REGION Network 3: Block description — Sections 4 to 10
   // ▄▄▄▄▄▄▄▄▄▄▄▄▄▄▄▄▄▄▄▄▄▄▄▄▄▄▄▄▄▄▄▄▄▄▄▄▄▄▄▄▄▄▄▄
   // 4.     Supervisory system interface
   // 
   // 
   // There is no supervisory system interface for this block. It is a debug simulation module and as 
   // such has no graphical symbol, block icon or faceplate.
   // 
   // 
   //                ━━━   ⬙⬙⬙⬙⬙⬙   ━━━
   // 
   // 
   // 
   // ▄▄▄▄▄▄▄▄▄▄▄▄▄▄▄▄▄▄▄▄▄▄▄▄▄▄▄▄▄▄▄▄▄▄▄▄▄▄▄▄▄▄▄▄
   // 5.     PARAMETERS
   // 
   // 
   // The following parameters are associated with the block:
   // 
   //  
   //  ――――――――――――――――――――――――――――――――――――――――――
   //  PARAM         FUNCTION                    TYPE      IN-OUT 
   //  ――――――――――――――――――――――――――――――――――――――――――
   //  SYS_SIGNALS      Common system signals              UT21000    In
   //           logic and timing signals for parametric access
   // 
   //  TRIGGER       Activates the simulation (the simulation will run     Bool      In
   //           whilever this signal is high), the elapsed time 
   //           is measured from the rising edge of this signal
   // 
   //  INPUT        The input time function, x(t) in the calculations     Real      In
   // 
   //  DYNAMIC_DATA      Data structure that holds the live data for the       UT39511    InOut
   //           simulation (damping factor, natural frequency, 
   //           system gain, elapsed time &c.)
   // 
   //  OUTPUT       The output time response, y(t) in the calculations   Real      Out
   //  ――――――――――――――――――――――――――――――――――――――――――
   // 
   //                ━━━   ⬙⬙⬙⬙⬙⬙   ━━━
   // 
   // 
   // 
   // ▄▄▄▄▄▄▄▄▄▄▄▄▄▄▄▄▄▄▄▄▄▄▄▄▄▄▄▄▄▄▄▄▄▄▄▄▄▄▄▄▄▄▄▄
   // 6.     DATA STRUCTURES AND USAGE
   // 
   // 
   // The block has the following associated data structure:
   // 
   // 
   //  ――――――――――――――――――――――――――――――――――――――――――
   //  DATA STRUCTURE             DESCRIPTION
   //  ――――――――――――――――――――――――――――――――――――――――――
   //  UT01000_St_SysRevision          Revision information for this block    See FC01001
   //  UT01001_St_SysLicence           Licence information for this block  See FC01001
   //  UT21000_Dy_SysSignals           System signals for logic and timing  See FC01001
   // 
   //  UT39511_Dy_DebugInst1Order        Dynamic data storage, contains live data, such as 
   //                     calculation variables, elapsed time, oscillation 
   //                     frequency and status signals
   //  ――――――――――――――――――――――――――――――――――――――――――
   // 
   // 
   // ▂▂▂▂▂▂▂▂▂▂▂▂▂▂▂▂▂▂▂▂▂▂▂▂▂▂▂▂▂▂▂▂▂▂▂▂▂▂▂▂▂▂▂▂
   // 6.1      UT39511_Dy_DebugInst1Order
   // 
   // The static data structure for an isolating valve.
   // 
   // 
   // 
   //  UT39511_Dy_DebugInst1Order (full contents)
   //  ――――――――――――――――――――――――――――――――――――――――――
   //  SIGNAL NAME          FUNCTION                     TYPE
   //  ――――――――――――――――――――――――――――――――――――――――――
   //  k_Gain             CONSTANT — Simulation system gain        Real
   //  k_TimeConstant        CONSTANT — The system time constant τ (s)       Real
   // 
   //  status_Running      STATUS — Simulation is running  Bool
   //                      (1 = running, 0 = stopped)
   //  status_Stopped        STATUS — Simulation is stopped (not running)    Bool
   //                      (1 = stopped, 0 = running)
   //  status_SteadyState     STATUS — Response is at steady state value             Bool
   //                      (1 = stead state reached ±2%)
   //  status_Aut           STATUS — Simulation is in automatic mode      Bool
   //                      (1 = automatic, 0 = manual)
   //  status_Man          STATUS — Simulation is in manual mode        Bool
   //                      (1 = manual, 0 = automatic)
   // 
   //  cal_TimeSteady        CALC — Time to reach steady state (s)       Real
   //                    zero for unstable response
   // 
   //  mode_AutMan       MODE — Automatic/manual mode selection     Bool
   //                      (1 = auto mode, 0 = manual mode)
   //  mode_ManTime       MODE — Manual mode time value (s)        Real
   // 
   //  actual_Output       ACTUAL — Output signal, same as OUTPUT param    Real
   //                      (y(t) or y[n])
   //  actual_PrevOutput      ACTUAL — Output value from the previous iteration    Real
   //                      (y[n-1])
   //  actual_StartTime         ACTUAL — CPU time when simulation started       DTL
   //  actual_Time        ACTUAL — CPU time of this iteration of simulation  DTL
   //  actual_PrevTime       ACTUAL — CPU time of last iteration of simulation     DTL
   //  actual_RunTime        ACTUAL — Elapsed time since the            Real
   //                      simulation started (s)
   //  actual_DeltaTime        ACTUAL — Time between this and last iteration (s)   Real
   //  ――――――――――――――――――――――――――――――――――――――――――
   // 
   // 
   //                ━━━   ⬙⬙⬙⬙⬙⬙   ━━━
   // 
   // 
   // 
   // ▄▄▄▄▄▄▄▄▄▄▄▄▄▄▄▄▄▄▄▄▄▄▄▄▄▄▄▄▄▄▄▄▄▄▄▄▄▄▄▄▄▄▄▄
   // 7.     CONSTANTS AND TEMPORARY (LOCAL) DATA
   // 
   // 
   // 
   // ▂▂▂▂▂▂▂▂▂▂▂▂▂▂▂▂▂▂▂▂▂▂▂▂▂▂▂▂▂▂▂▂▂▂▂▂▂▂▂▂▂▂▂▂
   // 7.1     Constants
   // 
   // 
   // The following constants data is used:
   // 
   //  ――――――――――――――――――――――――――――――――――――――――――
   //  SIGNAL NAME       Value     FUNCTION                 TYPE
   //  ――――――――――――――――――――――――――――――――――――――――――
   //  k_NEG_MAX       3.4E-38    Largest negative REAL number         Real
   //  ――――――――――――――――――――――――――――――――――――――――――
   // 
   // 
   // 
   // ▂▂▂▂▂▂▂▂▂▂▂▂▂▂▂▂▂▂▂▂▂▂▂▂▂▂▂▂▂▂▂▂▂▂▂▂▂▂▂▂▂▂▂▂
   // 7.2     Temporary (local) data
   // 
   // 
   // The following temporary data is used:
   // 
   //  ――――――――――――――――――――――――――――――――――――――――――
   //  SIGNAL NAME          FUNCTION                  TYPE
   //  ――――――――――――――――――――――――――――――――――――――――――
   //  revInfo             Revision information for the block         UT01000
   //  licInfo           Licensing information for the block      UT01001
   //  act_CPUTime           Current CPU time (this block call)       DTL
   //  cal_01          Partial calculation see § 3.4 for details      Real
   //  cal_02          Partial calculation see § 3.4 for details      Real
   //  cal_03          Partial calculation see § 3.4 for details      Real
   //  cal_04          Partial calculation see § 3.4 for details      Real
   //  cal_05          Partial calculation see § 3.4 for details      Real
   //  cal_06          Partial calculation see § 3.4 for details      Real
   //  wrkElapsedTime          Working storage area (current elapsed time)    LTIme
   //  wrkDeltaTime         Working storage area (current delta time)   LTIme
   //  wrkInt           Working storage area (integer)          Int
   //  wrkLInt            Working storage area (long integer)        ULInt
   //  wrkReal           Working storage (Real)             Real
   //  ――――――――――――――――――――――――――――――――――――――――――
   // 
   // 
   //                ━━━   ⬙⬙⬙⬙⬙⬙   ━━━
   // 
   // 
   // 
   // ▄▄▄▄▄▄▄▄▄▄▄▄▄▄▄▄▄▄▄▄▄▄▄▄▄▄▄▄▄▄▄▄▄▄▄▄▄▄▄▄▄▄▄▄
   // 8.     BLOCK CALLS AND ASSOCIATIONS
   // 
   // 
   // This section details any blocks which may be called from within this software module (subroutine 
   // functions for example), any partner blocks with which it may be associated (for example a 
   // receive module that is partner with a transmit module &c.). It lists any system functions which 
   // may be called (e.g. reading the real time clock) and any system data types that may be used.
   // 
   // Finally, it lists any special calling requirements for the block (for example, must be called from 
   // within a cyclic interrupt organisation block) and if the block is using “optimised access” (this is 
   // the default arrangement).
   // 
   // 
   // 
   // ▂▂▂▂▂▂▂▂▂▂▂▂▂▂▂▂▂▂▂▂▂▂▂▂▂▂▂▂▂▂▂▂▂▂▂▂▂▂▂▂▂▂▂▂
   // 8.1     Block calls from within this module
   // 
   // 
   // There are no PAL block calls from within this block.
   // 
   // 
   // 
   // ▂▂▂▂▂▂▂▂▂▂▂▂▂▂▂▂▂▂▂▂▂▂▂▂▂▂▂▂▂▂▂▂▂▂▂▂▂▂▂▂▂▂▂▂
   // 8.2     Blocks associated with this module
   // 
   // 
   // This is a stand-alone block and is not associated with any other blocks.
   // 
   // 
   // 
   // ▂▂▂▂▂▂▂▂▂▂▂▂▂▂▂▂▂▂▂▂▂▂▂▂▂▂▂▂▂▂▂▂▂▂▂▂▂▂▂▂▂▂▂▂
   // 8.3     System block calls and system data types
   // 
   // The following calls are made to system blocks:
   // 
   // 
   //  System block calls
   //  ――――――――――――――――――――――――――――――――――――――――――
   //  BLOCK          TITLE             DESCRIPTION  
   //  ――――――――――――――――――――――――――――――――――――――――――
   //  RD_LOC_T             Read the local RTC time    Reads the CPU real time clock 
   //  ――――――――――――――――――――――――――――――――――――――――――
   // 
   // There are no special system data types used.
   // 
   // 
   //                ━━━   ⬙⬙⬙⬙⬙⬙   ━━━
   // 
   // 
   // 
   // ▂▂▂▂▂▂▂▂▂▂▂▂▂▂▂▂▂▂▂▂▂▂▂▂▂▂▂▂▂▂▂▂▂▂▂▂▂▂▂▂▂▂▂▂
   // 8.4     Special properties and requirements
   // 
   // 
   // 
   // ▁▁▁▁▁▁▁▁▁▁▁▁▁▁▁▁▁▁▁▁▁▁▁▁▁▁▁▁▁▁▁▁▁▁▁▁▁▁▁▁▁▁▁▁
   // 8.4.1     Block optimisation, IEC compatibility and library conformance
   // 
   // 
   //    •   Block optimisation is ACTIVE for this block.
   // 
   //    •   The block has been checked for IEC compatibility and is compliant.
   // 
   //    •   The block is compatible with all IEC library-conformance module constraints
   // 
   // 
   // 
   // ▁▁▁▁▁▁▁▁▁▁▁▁▁▁▁▁▁▁▁▁▁▁▁▁▁▁▁▁▁▁▁▁▁▁▁▁▁▁▁▁▁▁▁▁
   // 8.4.2     Calling requirements
   // 
   // 
   // There are no special calling requirements for this block.
   // 
   //                ━━━   ⬙⬙⬙⬙⬙⬙   ━━━
   // 
   // 
   // 
   // ▄▄▄▄▄▄▄▄▄▄▄▄▄▄▄▄▄▄▄▄▄▄▄▄▄▄▄▄▄▄▄▄▄▄▄▄▄▄▄▄▄▄▄▄
   // 9.     EXAMPLE USAGE
   // 
   // 
   // The following shows a typical deployment of FC19512:
   // 
   //                         ┌─────────────
   //      ───────────────────┤ FC19511
   //                         ├───────────────┤
   //    "DB21001_DY_StdGlobalData".SysSignals ─┤ SYS_SIGNALS                  %MD910 
   //                         │               OUTPUT ├─  "SIM001_OUTPUT"
   //                         │               │
   //                                                        "1.0" ─┤ INPUT                     │
   //                         │               │
   //                   %M999.0     │               │
   //                  "SIM001_TRIG" ─┤ TRIGGER                     │
   //                         │               │
   //                         │
   //      "DB39511_Dy_DebugInst1Order".SIM001 ─┤ DYNAMIC_DATA
   //                         │
   //                         │
   //                                         │
   //                                ─────────┘
   // 
   // 
   //               ━━━   ⬙⬙⬙⬙⬙⬙   ━━━
   // 
   // 
   // 
   // ▄▄▄▄▄▄▄▄▄▄▄▄▄▄▄▄▄▄▄▄▄▄▄▄▄▄▄▄▄▄▄▄▄▄▄▄▄▄▄▄▄▄▄▄
   // 10.     TEST AND VERIFICATION PATH
   // 
   // 
   // The following diagram shows the full test and verification path for the formal release of each 
   // version of the software module. See the Test Plan [Ref. 003] for full details, available here:
   //         https://psop.uk/pal-tp-p
   // 
   // 
   //         FC19151-T001
   // 
   //     Test version: 000.801  
   //  Released version: 001.000   
   // Released commit: D0017    
   // 
   //        SCR      SMT 
   // ＿＿＿＿＿＿┌┐＿＿ ▛▜ ＿
   //       └┘   ▙▟  
   // Initial test           
   // 
   // Initial test to release the      
   // module following the      
   // development stage.       
   // Full SMT              
   // 
   // 
   // Where:
   // ――――――――――――――――――――――――――――――――――――――――――――
   //  SCR    Source Code Review      A visual inspection of the software to ensure it has been written  
   // ┌┐             to the correct standards, uses the correct structures within the
   // └┘             software and is generally suitable for deployment.               
   // 
   //  SMT Software Module Test    A full and detailed test of an individual software module in
   //   ▛▜              isolation; such testing requires that all branches of the 
   //   ▙▟              software are tested. 
   // 
   //                It tests all the interfaces to the module, any data recorded or 
   //                stored by the module, all error and exception handling functions 
   //                and tests all timed and interrupt driven operations.
   // 
   //  SCV Software Compatibility     A mechanism for verifying that no executable code software 
   // ╓╖    Verification          changes have been made to a module following changes to
   // ╙╜             comment fields.
   // 
   //                Allows typographical errors &c. to be corrected without forcing 
   //                a full SMT on a module that has not functionally changed.
   // ――――――――――――――――――――――――――――――――――――――――――――
   // 
   // An SCV can only be performed on a module that has at some point previously, successfully 
   // completed both an SCR and SMT. Where an SCV is implemented, it replaces the requirement for 
   // both the SCR and the SMT for the test iteration in question.
   // 
   //                ━━━   ⬙⬙⬙⬙⬙⬙   ━━━
   // 
   // 
   // ██████████████ █ █ █ █  END   █ █ █ █ ██████████████
END_REGION

REGION Network 4: Current revision and modification history
   // ▄▄▄▄▄▄▄▄▄▄▄▄▄▄▄▄▄▄▄▄▄▄▄▄▄▄▄▄▄▄▄▄▄▄▄▄▄▄▄▄▄▄▄▄
   // MODIFICATION HISTORY
   // 
   // 
   // The revision data shown here, in the network comments, contains additional information 
   // reflecting the software development workflow under the version control system (VCS) employed 
   // to track all software changes.
   // 
   // The VCS in use is the Git Source Code Management system in conjunction with the GitHub online 
   // hosting system. The software in its entirety is available in the GitHub remote repository:
   // 
   //      https://github.com/practicalseries/PS2001-pal-software
   // 
   // The repository is public and can be freely copied (forked in GitHub terminology) and used 
   // under the MIT licence. 
   // 
   // The MIT licence is reproduced in full in the last network of this software module.
   // 
   // 
   //  ―――――――――――――――――――――――――――――――――――――――――――
   //  DATE       REVISION             MASTER BRANCH     DEV
   //          (nnn.amm)   COMMIT TAG    (Base ---> Merge)    BRANCH   Author
   //  ———————————————————————————————————————————
   //  2023.02.26    000.101   D0016A-000.101   D0016 N/A     D0016A   M. Gledhill
   //                        FC19511 Block created — Comments added
   //  ———————————————————————————————————————————
   //   Where: nnn  =  Major revision
   //         a  =  Type (1-7 Development, 8 Proving, 9 Qualification, 0 Release)
   //       mm  =  Minor revision (must be 00 if a = 0)
   //         Block properties version number should be set to nn.a (only one decimal place)
   // 
   // ▄▄▄▄▄▄▄▄▄▄▄▄▄▄▄▄▄▄▄▄▄▄▄▄▄▄▄▄▄▄▄▄▄▄▄▄▄▄▄▄▄▄▄▄
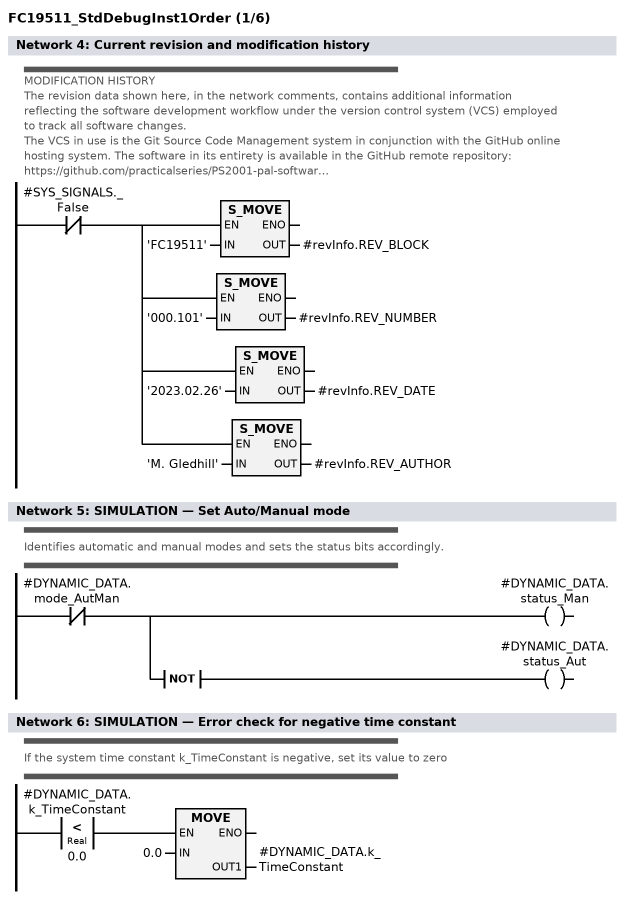
   RUNG wire#powerrail
      I_Contact( #SYS_SIGNALS._False )
      wire#w1
      S_Move(in := 'FC19511', out => #revInfo.REV_BLOCK)
   END_RUNG
   RUNG wire#w1
      S_Move(in := '000.101', out => #revInfo.REV_NUMBER)
   END_RUNG
   RUNG wire#w1
      S_Move(in := '2023.02.26', out => #revInfo.REV_DATE)
   END_RUNG
   RUNG wire#w1
      S_Move(in := 'M. Gledhill', out => #revInfo.REV_AUTHOR)
   END_RUNG
   // the same network as SCL:
   IF NOT #SYS_SIGNALS._False THEN
       #revInfo.REV_BLOCK := 'FC19511';
       #revInfo.REV_NUMBER := '000.101';
       #revInfo.REV_DATE := '2023.02.26';
       #revInfo.REV_AUTHOR := 'M. Gledhill';
   END_IF;
END_REGION

REGION Network 5: SIMULATION — Set Auto/Manual mode
   // ▀▀▀▀▀▀▀▀▀▀▀▀▀▀▀▀▀▀▀▀▀▀▀▀▀▀▀▀▀▀▀▀▀▀▀▀▀▀▀▀▀▀▀▀
   // Identifies automatic and manual modes and sets the status bits accordingly.
   // ▄▄▄▄▄▄▄▄▄▄▄▄▄▄▄▄▄▄▄▄▄▄▄▄▄▄▄▄▄▄▄▄▄▄▄▄▄▄▄▄▄▄▄▄
   RUNG wire#powerrail
      I_Contact( #DYNAMIC_DATA.mode_AutMan )
      wire#w1
      Coil( #DYNAMIC_DATA.status_Man )
   END_RUNG
   RUNG wire#w1
      Not()
      Coil( #DYNAMIC_DATA.status_Aut )
   END_RUNG
   // the same network as SCL:
   #DYNAMIC_DATA.status_Man := NOT #DYNAMIC_DATA.mode_AutMan;
   #DYNAMIC_DATA.status_Aut := NOT (NOT #DYNAMIC_DATA.mode_AutMan);
END_REGION

REGION Network 6: SIMULATION — Error check for negative time constant
   // ▀▀▀▀▀▀▀▀▀▀▀▀▀▀▀▀▀▀▀▀▀▀▀▀▀▀▀▀▀▀▀▀▀▀▀▀▀▀▀▀▀▀▀▀
   // If the system time constant k_TimeConstant is negative, set its value to zero
   // ▄▄▄▄▄▄▄▄▄▄▄▄▄▄▄▄▄▄▄▄▄▄▄▄▄▄▄▄▄▄▄▄▄▄▄▄▄▄▄▄▄▄▄▄
   RUNG wire#powerrail
      { S7_Templates := "SrcType := Real" } LT_Contact(in1 := #DYNAMIC_DATA.k_TimeConstant, in2 := 0.0)
      Move(in := 0.0, out1 => #DYNAMIC_DATA.k_TimeConstant)
   END_RUNG
   // the same network as SCL:
   IF #DYNAMIC_DATA.k_TimeConstant < 0.0 THEN #DYNAMIC_DATA.k_TimeConstant := 0.0; END_IF;
END_REGION

REGION Network 7: SIMULATION INACTIVE — Reset data — Block end
   // ▀▀▀▀▀▀▀▀▀▀▀▀▀▀▀▀▀▀▀▀▀▀▀▀▀▀▀▀▀▀▀▀▀▀▀▀▀▀▀▀▀▀▀▀
   // If the simulation is not running (TRIGGER = 0), set status to stopped and reset all calculated data
   // and status signals.
   // 
   // Set the previous time to the current CPU time (in readiness for the start of the simulation)
   // 
   // Set the OUTPUT, actual_Output and actual_PrevOutput to zero
   // 
   // If the simulation is not running, the block will terminate at this point.
   // ▄▄▄▄▄▄▄▄▄▄▄▄▄▄▄▄▄▄▄▄▄▄▄▄▄▄▄▄▄▄▄▄▄▄▄▄▄▄▄▄▄▄▄▄
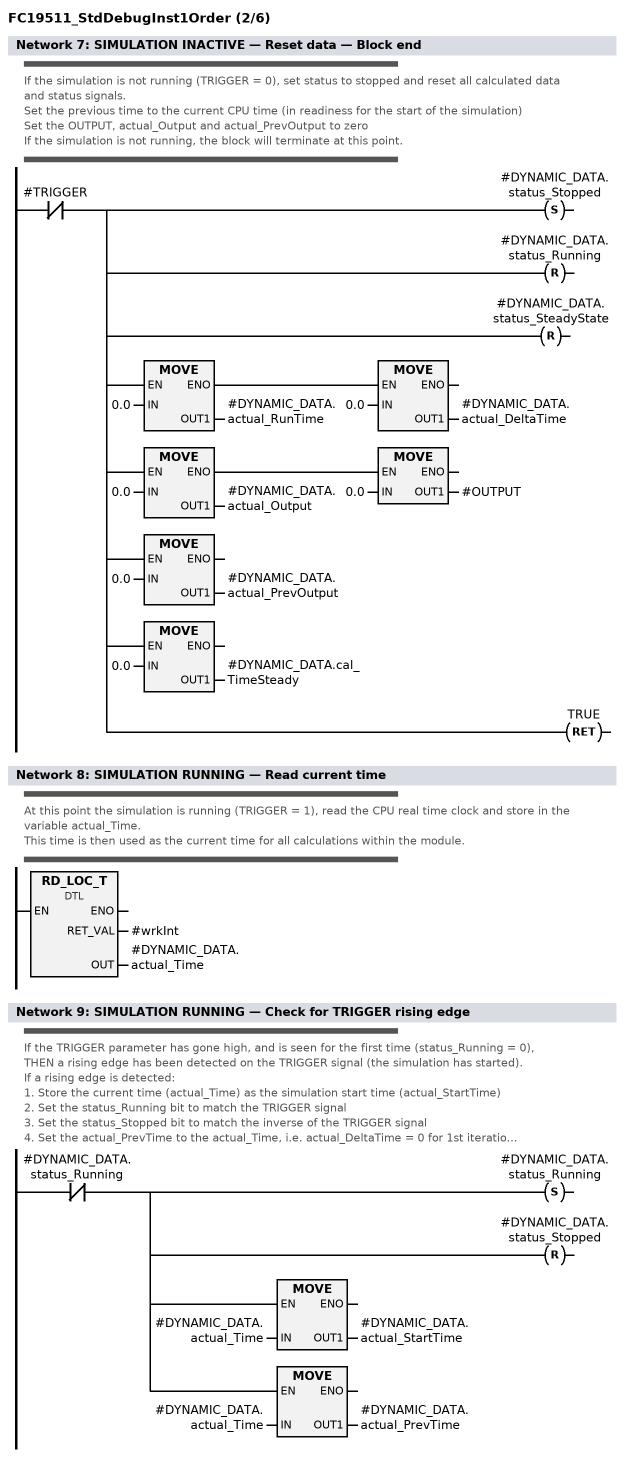
   IF NOT #TRIGGER THEN
       #DYNAMIC_DATA.status_Stopped := TRUE;
       #DYNAMIC_DATA.status_Running := FALSE;
       #DYNAMIC_DATA.status_SteadyState := FALSE;
       #DYNAMIC_DATA.actual_RunTime := 0.0;
       #DYNAMIC_DATA.actual_DeltaTime := 0.0;
       #DYNAMIC_DATA.actual_Output := 0.0;
       #OUTPUT := 0.0;
       #DYNAMIC_DATA.actual_PrevOutput := 0.0;
       #DYNAMIC_DATA.cal_TimeSteady := 0.0;
       ENO := TRUE;
       RETURN;
   END_IF;
END_REGION

REGION Network 8: SIMULATION RUNNING — Read current time
   // ▀▀▀▀▀▀▀▀▀▀▀▀▀▀▀▀▀▀▀▀▀▀▀▀▀▀▀▀▀▀▀▀▀▀▀▀▀▀▀▀▀▀▀▀
   // At this point the simulation is running (TRIGGER = 1), read the CPU real time clock and store in the 
   // variable actual_Time.
   // 
   // This time is then used as the current time for all calculations within the module.
   // ▄▄▄▄▄▄▄▄▄▄▄▄▄▄▄▄▄▄▄▄▄▄▄▄▄▄▄▄▄▄▄▄▄▄▄▄▄▄▄▄▄▄▄▄
   RUNG wire#powerrail
      { S7_Templates := "date_type := DTL" } RD_LOC_T(RET_VAL => #wrkInt, OUT => #DYNAMIC_DATA.actual_Time)
   END_RUNG
   // the same network as SCL:
   #wrkInt := RD_LOC_T(OUT => #DYNAMIC_DATA.actual_Time);
END_REGION

REGION Network 9: SIMULATION RUNNING — Check for TRIGGER rising edge
   // ▀▀▀▀▀▀▀▀▀▀▀▀▀▀▀▀▀▀▀▀▀▀▀▀▀▀▀▀▀▀▀▀▀▀▀▀▀▀▀▀▀▀▀▀
   // If the TRIGGER parameter has gone high, and is seen for the first time (status_Running = 0),
   // THEN a rising edge has been detected on the TRIGGER signal (the simulation has started).
   // 
   // If a rising edge is detected:
   //   1. Store the current time (actual_Time) as the simulation start time (actual_StartTime)
   //   2. Set the status_Running bit to match the TRIGGER signal
   //   3. Set the status_Stopped bit to match the inverse of the TRIGGER signal
   //   4. Set the actual_PrevTime to the actual_Time, i.e. actual_DeltaTime = 0 for 1st iteration
   // ▄▄▄▄▄▄▄▄▄▄▄▄▄▄▄▄▄▄▄▄▄▄▄▄▄▄▄▄▄▄▄▄▄▄▄▄▄▄▄▄▄▄▄▄
   RUNG wire#powerrail
      I_Contact( #DYNAMIC_DATA.status_Running )
      wire#w1
      S_Coil( #DYNAMIC_DATA.status_Running )
   END_RUNG
   RUNG wire#w1
      R_Coil( #DYNAMIC_DATA.status_Stopped )
   END_RUNG
   RUNG wire#w1
      Move(in := #DYNAMIC_DATA.actual_Time, out1 => #DYNAMIC_DATA.actual_StartTime)
   END_RUNG
   RUNG wire#w1
      Move(in := #DYNAMIC_DATA.actual_Time, out1 => #DYNAMIC_DATA.actual_PrevTime)
   END_RUNG
   // the same network as SCL:
   #_w1 := NOT #DYNAMIC_DATA.status_Running;
   IF #_w1 THEN
       #DYNAMIC_DATA.status_Running := TRUE;
       #DYNAMIC_DATA.status_Stopped := FALSE;
       #DYNAMIC_DATA.actual_StartTime := #DYNAMIC_DATA.actual_Time;
       #DYNAMIC_DATA.actual_PrevTime := #DYNAMIC_DATA.actual_Time;
   END_IF;
END_REGION

REGION Network 10: SIMULATION RUNNING — Calculate current elapsed time
   // ▀▀▀▀▀▀▀▀▀▀▀▀▀▀▀▀▀▀▀▀▀▀▀▀▀▀▀▀▀▀▀▀▀▀▀▀▀▀▀▀▀▀▀▀
   // If the TRIGGER parameter is high (the simulation is running), then:
   // Subtract the start time from the current time to give the current elapsed time (wrkElapsedTime)
   // 
   // The elapsed time is calculated in the LTIme format
   // ▄▄▄▄▄▄▄▄▄▄▄▄▄▄▄▄▄▄▄▄▄▄▄▄▄▄▄▄▄▄▄▄▄▄▄▄▄▄▄▄▄▄▄▄
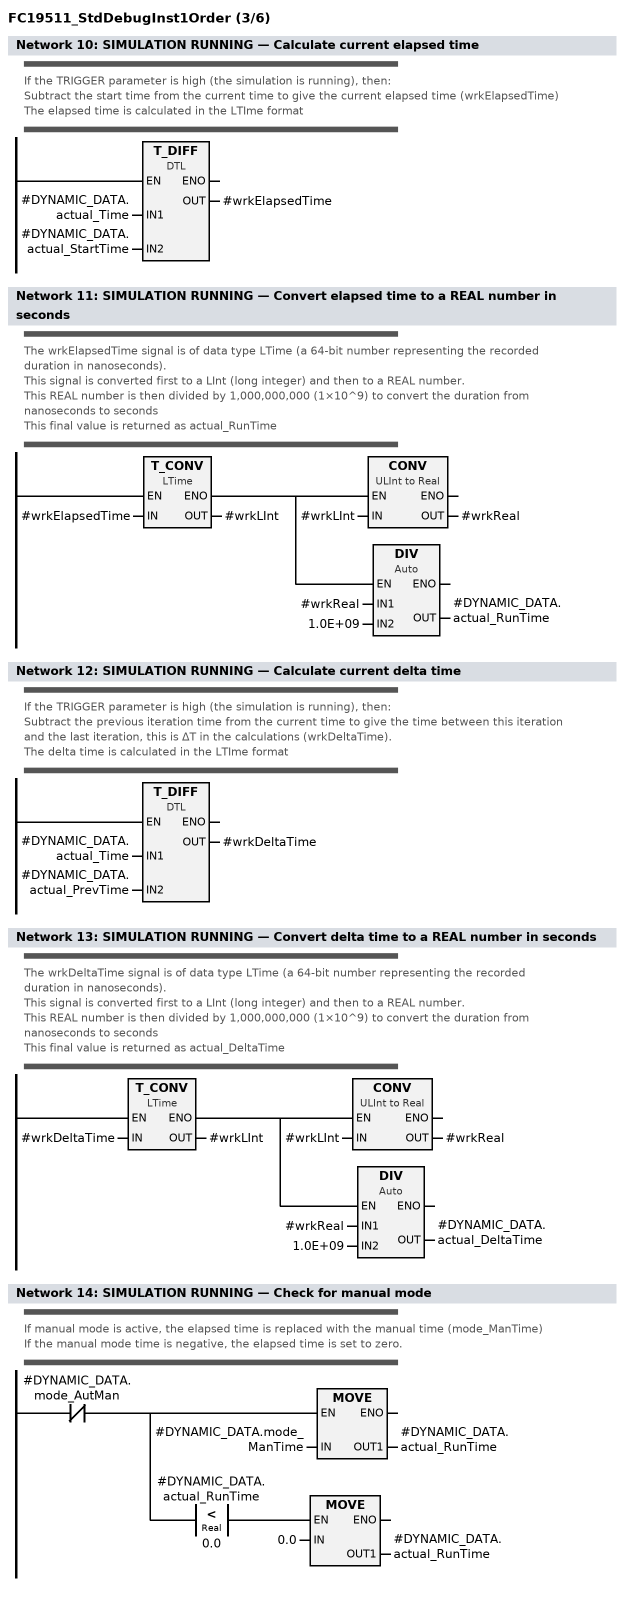
   RUNG wire#powerrail
      { S7_Templates := "[date_type := DTL, time_type := LTime]" } T_DIFF(IN1 := #DYNAMIC_DATA.actual_Time, IN2 := #DYNAMIC_DATA.actual_StartTime, OUT => #wrkElapsedTime)
   END_RUNG
   // the same network as SCL:
   T_DIFF(IN1 := #DYNAMIC_DATA.actual_Time, IN2 := #DYNAMIC_DATA.actual_StartTime, OUT => #wrkElapsedTime);
END_REGION

REGION Network 11: SIMULATION RUNNING — Convert elapsed time to a REAL number in seconds
   // ▀▀▀▀▀▀▀▀▀▀▀▀▀▀▀▀▀▀▀▀▀▀▀▀▀▀▀▀▀▀▀▀▀▀▀▀▀▀▀▀▀▀▀▀
   // The wrkElapsedTime signal is of data type LTime (a 64-bit number representing the recorded
   // duration in nanoseconds).
   // 
   // This signal is converted first to a LInt (long integer) and then to a REAL number.
   // 
   // This REAL number is then divided by 1,000,000,000 (1×10^9) to convert the duration from 
   // nanoseconds to seconds
   // 
   // This final value is returned as actual_RunTime
   // ▄▄▄▄▄▄▄▄▄▄▄▄▄▄▄▄▄▄▄▄▄▄▄▄▄▄▄▄▄▄▄▄▄▄▄▄▄▄▄▄▄▄▄▄
   RUNG wire#powerrail
      { S7_Templates := "[src_type := LTime, dest_type := ULInt]" } T_CONV(IN := #wrkElapsedTime, OUT => #wrkLInt)
      wire#w1
      { S7_Templates := "[SrcType := ULInt, DestType := Real]" } Convert(in := #wrkLInt, out => #wrkReal)
   END_RUNG
   RUNG wire#w1
      Div(in1 := #wrkReal, in2 := 1.0E+09, out => #DYNAMIC_DATA.actual_RunTime)
   END_RUNG
   // the same network as SCL:
   T_CONV(IN := #wrkElapsedTime, OUT => #wrkLInt, ENO => #_w1);
   IF #_w1 THEN
       #wrkReal := ULINT_TO_REAL(#wrkLInt);
       #DYNAMIC_DATA.actual_RunTime := #wrkReal / 1.0E+09;
   END_IF;
END_REGION

REGION Network 12: SIMULATION RUNNING — Calculate current delta time
   // ▀▀▀▀▀▀▀▀▀▀▀▀▀▀▀▀▀▀▀▀▀▀▀▀▀▀▀▀▀▀▀▀▀▀▀▀▀▀▀▀▀▀▀▀
   // If the TRIGGER parameter is high (the simulation is running), then:
   // Subtract the previous iteration time from the current time to give the time between this iteration
   // and the last iteration, this is ΔT in the calculations (wrkDeltaTime).
   // 
   // The delta time is calculated in the LTIme format
   // ▄▄▄▄▄▄▄▄▄▄▄▄▄▄▄▄▄▄▄▄▄▄▄▄▄▄▄▄▄▄▄▄▄▄▄▄▄▄▄▄▄▄▄▄
   RUNG wire#powerrail
      { S7_Templates := "[date_type := DTL, time_type := LTime]" } T_DIFF(IN1 := #DYNAMIC_DATA.actual_Time, IN2 := #DYNAMIC_DATA.actual_PrevTime, OUT => #wrkDeltaTime)
   END_RUNG
   // the same network as SCL:
   T_DIFF(IN1 := #DYNAMIC_DATA.actual_Time, IN2 := #DYNAMIC_DATA.actual_PrevTime, OUT => #wrkDeltaTime);
END_REGION

REGION Network 13: SIMULATION RUNNING — Convert delta time to a REAL number in seconds
   // ▀▀▀▀▀▀▀▀▀▀▀▀▀▀▀▀▀▀▀▀▀▀▀▀▀▀▀▀▀▀▀▀▀▀▀▀▀▀▀▀▀▀▀▀
   // The wrkDeltaTime signal is of data type LTime (a 64-bit number representing the recorded
   // duration in nanoseconds).
   // 
   // This signal is converted first to a LInt (long integer) and then to a REAL number.
   // 
   // This REAL number is then divided by 1,000,000,000 (1×10^9) to convert the duration from 
   // nanoseconds to seconds
   // 
   // This final value is returned as actual_DeltaTime
   // ▄▄▄▄▄▄▄▄▄▄▄▄▄▄▄▄▄▄▄▄▄▄▄▄▄▄▄▄▄▄▄▄▄▄▄▄▄▄▄▄▄▄▄▄
   RUNG wire#powerrail
      { S7_Templates := "[src_type := LTime, dest_type := ULInt]" } T_CONV(IN := #wrkDeltaTime, OUT => #wrkLInt)
      wire#w1
      { S7_Templates := "[SrcType := ULInt, DestType := Real]" } Convert(in := #wrkLInt, out => #wrkReal)
   END_RUNG
   RUNG wire#w1
      Div(in1 := #wrkReal, in2 := 1.0E+09, out => #DYNAMIC_DATA.actual_DeltaTime)
   END_RUNG
   // the same network as SCL:
   T_CONV(IN := #wrkDeltaTime, OUT => #wrkLInt, ENO => #_w1);
   IF #_w1 THEN
       #wrkReal := ULINT_TO_REAL(#wrkLInt);
       #DYNAMIC_DATA.actual_DeltaTime := #wrkReal / 1.0E+09;
   END_IF;
END_REGION

REGION Network 14: SIMULATION RUNNING — Check for manual mode
   // ▀▀▀▀▀▀▀▀▀▀▀▀▀▀▀▀▀▀▀▀▀▀▀▀▀▀▀▀▀▀▀▀▀▀▀▀▀▀▀▀▀▀▀▀
   // If manual mode is active, the elapsed time is replaced with the manual time (mode_ManTime)
   // 
   // If the manual mode time is negative, the elapsed time is set to zero.
   // ▄▄▄▄▄▄▄▄▄▄▄▄▄▄▄▄▄▄▄▄▄▄▄▄▄▄▄▄▄▄▄▄▄▄▄▄▄▄▄▄▄▄▄▄
   RUNG wire#powerrail
      I_Contact( #DYNAMIC_DATA.mode_AutMan )
      wire#w1
      Move(in := #DYNAMIC_DATA.mode_ManTime, out1 => #DYNAMIC_DATA.actual_RunTime)
   END_RUNG
   RUNG wire#w1
      { S7_Templates := "SrcType := Real" } LT_Contact(in1 := #DYNAMIC_DATA.actual_RunTime, in2 := 0.0)
      Move(in := 0.0, out1 => #DYNAMIC_DATA.actual_RunTime)
   END_RUNG
   // the same network as SCL:
   #_w1 := NOT #DYNAMIC_DATA.mode_AutMan;
   IF #_w1 THEN #DYNAMIC_DATA.actual_RunTime := #DYNAMIC_DATA.mode_ManTime; END_IF;
   IF #_w1 AND (#DYNAMIC_DATA.actual_RunTime < 0.0) THEN #DYNAMIC_DATA.actual_RunTime := 0.0; END_IF;
END_REGION

REGION Network 15: SIMULATION RUNNING — Real-time simulation calculation
   // ▀▀▀▀▀▀▀▀▀▀▀▀▀▀▀▀▀▀▀▀▀▀▀▀▀▀▀▀▀▀▀▀▀▀▀▀▀▀▀▀▀▀▀▀
   // If the simulation is running and is in automatic mode, the following iterative, Real-time 
   // simulation calculation is carried out:
   // 
   // CALCULATION:
   //                               ΔT
   //    y[n] = Ka x[n]  ┼ (1-a) y[n-1]   where: a = ----------
   //                             τ+ΔT
   // 
   // Is rendered into the correct format as follows:
   // 
   // 
   //  cal_01 = ΔT             =  actual_DeltaTime
   // 
   //  cal_02 = τ + ΔT             = k_TimeConstant + cal_01
   // 
   //                ΔT
   //  cal_03 = a = ----------          = cal_01 ÷ cal_02
   //                 τ+ΔT
   // 
   //  cal_04 = 1 - a             = 1 - cal_03
   // 
   // 
   //  cal_05 = Kax[n]            = k_Gain × cal_03 × INPUT
   // 
   //  cal_06 = (1-a) y[n-1]          = cal_04 × actual_PrevOutput
   // 
   // 
   //  OUTPUT  = Ka x[n]  ┼ (1-a) y[n-1]      = cal_05 × cal_06
   // 
   // 
   // ▄▄▄▄▄▄▄▄▄▄▄▄▄▄▄▄▄▄▄▄▄▄▄▄▄▄▄▄▄▄▄▄▄▄▄▄▄▄▄▄▄▄▄▄
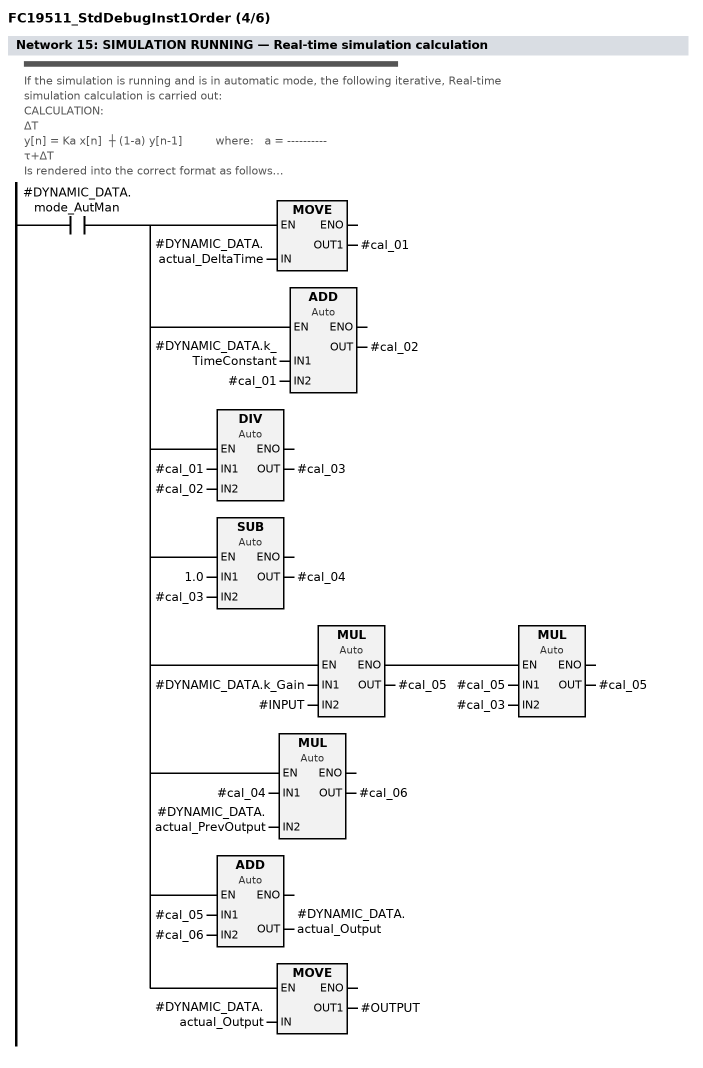
   RUNG wire#powerrail
      Contact( #DYNAMIC_DATA.mode_AutMan )
      wire#w1
      Move(in := #DYNAMIC_DATA.actual_DeltaTime, out1 => #cal_01)
   END_RUNG
   RUNG wire#w1
      Add(in1 := #DYNAMIC_DATA.k_TimeConstant, in2 := #cal_01, out => #cal_02)
   END_RUNG
   RUNG wire#w1
      Div(in1 := #cal_01, in2 := #cal_02, out => #cal_03)
   END_RUNG
   RUNG wire#w1
      Sub(in1 := 1.0, in2 := #cal_03, out => #cal_04)
   END_RUNG
   RUNG wire#w1
      Mul(in1 := #DYNAMIC_DATA.k_Gain, in2 := #INPUT, out => #cal_05)
      Mul(in1 := #cal_05, in2 := #cal_03, out => #cal_05)
   END_RUNG
   RUNG wire#w1
      Mul(in1 := #cal_04, in2 := #DYNAMIC_DATA.actual_PrevOutput, out => #cal_06)
   END_RUNG
   RUNG wire#w1
      Add(in1 := #cal_05, in2 := #cal_06, out => #DYNAMIC_DATA.actual_Output)
   END_RUNG
   RUNG wire#w1
      Move(in := #DYNAMIC_DATA.actual_Output, out1 => #OUTPUT)
   END_RUNG
   // the same network as SCL:
   IF #DYNAMIC_DATA.mode_AutMan THEN
       #cal_01 := #DYNAMIC_DATA.actual_DeltaTime;
       #cal_02 := #DYNAMIC_DATA.k_TimeConstant + #cal_01;
       #cal_03 := #cal_01 / #cal_02;
       #cal_04 := 1.0 - #cal_03;
       #cal_05 := #DYNAMIC_DATA.k_Gain * #INPUT;
       #cal_05 := #cal_05 * #cal_03;
       #cal_06 := #cal_04 * #DYNAMIC_DATA.actual_PrevOutput;
       #DYNAMIC_DATA.actual_Output := #cal_05 + #cal_06;
       #OUTPUT := #DYNAMIC_DATA.actual_Output;
   END_IF;
END_REGION

REGION Network 16: SIMULATION RUNNING — Over damped — Ancillary calculations
   // ▀▀▀▀▀▀▀▀▀▀▀▀▀▀▀▀▀▀▀▀▀▀▀▀▀▀▀▀▀▀▀▀▀▀▀▀▀▀▀▀▀▀▀▀
   // If the simulation is running and is in manual mode, the following discrete manual response to a 
   // step input calculation is carried out:
   // 
   // 
   // CALCULATION:
   // 
   //          ┌      -t/τ  ┐
   //    y(t) = KX│ 1 ─  e   │
   //          └       ┘
   // 
   // 
   // Is rendered into the correct format as follows:
   // 
   // 
   //  cal_01 =  -t/τ            = - 1 × actual_RunTime ÷  k_TimeConstant
   // 
   //          - t/τ
   //  cal_02 = ｅ              = EXP (cal_01)
   // 
   //                - t/τ
   //  cal_03 = 1 ─  ｅ              = 1 - cal_02
   // 
   // 
   //              ┌      -t/τ  ┐
   //  OUTPUT  = KX│ 1 ─  e   │       = k_Gain × INPUT × cal_03
   //              └       ┘
   // 
   // Note:    If k_TimeConstant = 0, cal_01 is set to the value k_NEG_MAX (the largest
   //      negative value available to a real number), preventing divide by zero errors.
   // 
   // ▄▄▄▄▄▄▄▄▄▄▄▄▄▄▄▄▄▄▄▄▄▄▄▄▄▄▄▄▄▄▄▄▄▄▄▄▄▄▄▄▄▄▄▄
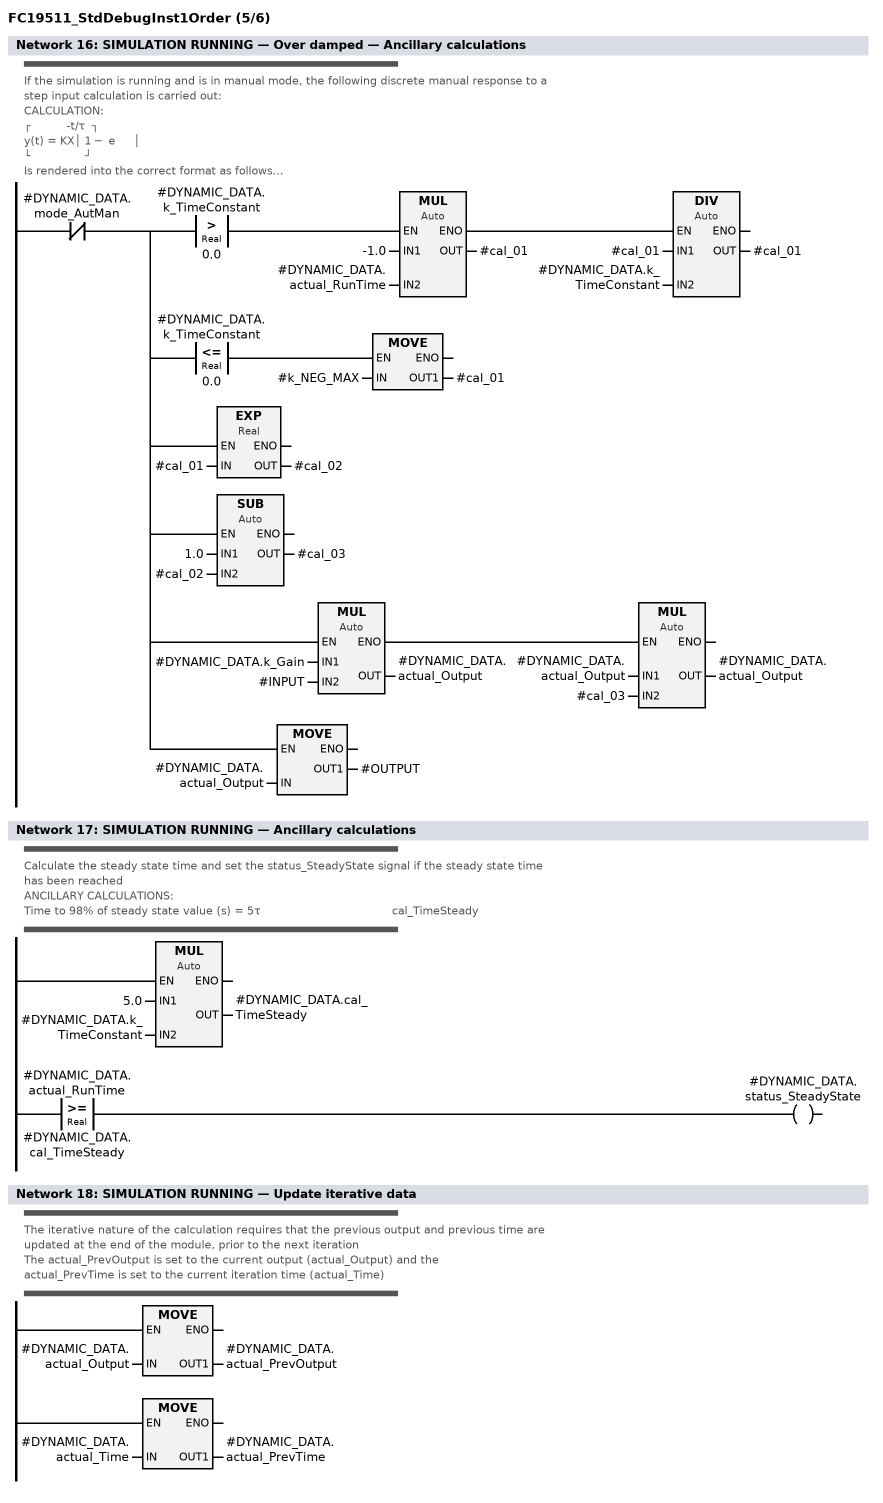
   #_w1 := NOT #DYNAMIC_DATA.mode_AutMan;
   IF #_w1 AND (#DYNAMIC_DATA.k_TimeConstant > 0.0) THEN
       #cal_01 := (-1.0) * #DYNAMIC_DATA.actual_RunTime;
       #cal_01 := #cal_01 / #DYNAMIC_DATA.k_TimeConstant;
   END_IF;
   IF #_w1 AND (#DYNAMIC_DATA.k_TimeConstant <= 0.0) THEN #cal_01 := #k_NEG_MAX; END_IF;
   IF #_w1 THEN
       #cal_02 := EXP(#cal_01);
       #cal_03 := 1.0 - #cal_02;
       #DYNAMIC_DATA.actual_Output := #DYNAMIC_DATA.k_Gain * #INPUT;
       #DYNAMIC_DATA.actual_Output := #DYNAMIC_DATA.actual_Output * #cal_03;
       #OUTPUT := #DYNAMIC_DATA.actual_Output;
   END_IF;
END_REGION

REGION Network 17: SIMULATION RUNNING — Ancillary calculations
   // ▀▀▀▀▀▀▀▀▀▀▀▀▀▀▀▀▀▀▀▀▀▀▀▀▀▀▀▀▀▀▀▀▀▀▀▀▀▀▀▀▀▀▀▀
   // Calculate the steady state time and set the status_SteadyState signal if the steady state time
   // has been reached
   // 
   // 
   // 
   // ANCILLARY CALCULATIONS:
   // 
   //  Time to 98% of steady state value (s) = 5τ              cal_TimeSteady
   // ▄▄▄▄▄▄▄▄▄▄▄▄▄▄▄▄▄▄▄▄▄▄▄▄▄▄▄▄▄▄▄▄▄▄▄▄▄▄▄▄▄▄▄▄
   RUNG wire#powerrail
      Mul(in1 := 5.0, in2 := #DYNAMIC_DATA.k_TimeConstant, out => #DYNAMIC_DATA.cal_TimeSteady)
   END_RUNG
   RUNG wire#powerrail
      { S7_Templates := "SrcType := Real" } GE_Contact(in1 := #DYNAMIC_DATA.actual_RunTime, in2 := #DYNAMIC_DATA.cal_TimeSteady)
      Coil( #DYNAMIC_DATA.status_SteadyState )
   END_RUNG
   // the same network as SCL:
   #DYNAMIC_DATA.cal_TimeSteady := 5.0 * #DYNAMIC_DATA.k_TimeConstant;
   #DYNAMIC_DATA.status_SteadyState := #DYNAMIC_DATA.actual_RunTime >= #DYNAMIC_DATA.cal_TimeSteady;
END_REGION

REGION Network 18: SIMULATION RUNNING — Update iterative data
   // ▀▀▀▀▀▀▀▀▀▀▀▀▀▀▀▀▀▀▀▀▀▀▀▀▀▀▀▀▀▀▀▀▀▀▀▀▀▀▀▀▀▀▀▀
   // The iterative nature of the calculation requires that the previous output and previous time are
   // updated at the end of the module, prior to the next iteration
   // 
   // The actual_PrevOutput is set to the current output (actual_Output) and the
   // actual_PrevTime is set to the current iteration time (actual_Time)
   // ▄▄▄▄▄▄▄▄▄▄▄▄▄▄▄▄▄▄▄▄▄▄▄▄▄▄▄▄▄▄▄▄▄▄▄▄▄▄▄▄▄▄▄▄
   RUNG wire#powerrail
      Move(in := #DYNAMIC_DATA.actual_Output, out1 => #DYNAMIC_DATA.actual_PrevOutput)
   END_RUNG
   RUNG wire#powerrail
      Move(in := #DYNAMIC_DATA.actual_Time, out1 => #DYNAMIC_DATA.actual_PrevTime)
   END_RUNG
   // the same network as SCL:
   #DYNAMIC_DATA.actual_PrevOutput := #DYNAMIC_DATA.actual_Output;
   #DYNAMIC_DATA.actual_PrevTime := #DYNAMIC_DATA.actual_Time;
END_REGION

REGION Network 19: LICENCE AND CONTACT INFORMATION
   // ▀▀▀▀▀▀▀▀▀▀▀▀▀▀▀▀▀▀▀▀▀▀▀▀▀▀▀▀▀▀▀▀▀▀▀▀▀▀▀▀▀▀▀▀
   // LICENCE AND CONTACT INFORMATION
   // 
   // This software and its associated documentation is made available under the MIT Licence:
   // 
   // ════════════════════════════════════════════
   // 
   // The MIT License (MIT)
   // 
   // Copyright © 2020 Michael Gledhill
   // 
   // Permission is hereby granted, free of charge, to any person obtaining a copy of this software 
   // and associated documentation files (the “Software”), to deal in the Software without restriction, 
   // including without limitation the rights to use, copy, modify, merge, publish, distribute, 
   // sublicense, and/or sell copies of the Software, and to permit persons to whom the Software is 
   // furnished to do so, subject to the following conditions: 
   // 
   // The above copyright notice and this permission notice shall be included in all copies or 
   // substantial portions of the Software.
   // 
   // THE SOFTWARE IS PROVIDED “AS IS”, WITHOUT WARRANTY OF ANY KIND, EXPRESS OR IMPLIED, 
   // INCLUDING BUT NOT LIMITED TO THE WARRANTIES OF MERCHANTABILITY, FITNESS FOR A 
   // PARTICULAR PURPOSE AND NON-INFRINGEMENT. IN NO EVENT SHALL THE AUTHORS OR COPYRIGHT 
   // HOLDERS BE LIABLE FOR ANY CLAIM, DAMAGES OR OTHER LIABILITY, WHETHER IN AN ACTION OF 
   // CONTRACT, TORT OR OTHERWISE, ARISING FROM, OUT OF OR IN CONNECTION WITH THE SOFTWARE 
   // OR THE USE OR OTHER DEALINGS IN THE SOFTWARE.
   // 
   // ════════════════════════════════════════════
   //                    ┌────────────┐
   // You can reach the author by email here:   │  mg@practicalseries.com  │
   //                    └────────────┘
   // Questions, corrections, constructive criticism and complaints (polite ones) are invited.
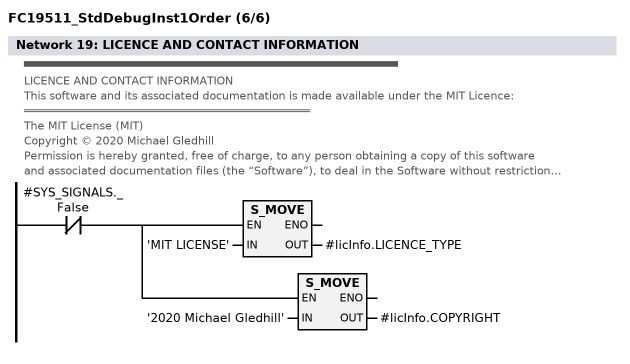
   RUNG wire#powerrail
      I_Contact( #SYS_SIGNALS._False )
      wire#w1
      S_Move(in := 'MIT LICENSE', out => #licInfo.LICENCE_TYPE)
   END_RUNG
   RUNG wire#w1
      S_Move(in := '2020 Michael Gledhill', out => #licInfo.COPYRIGHT)
   END_RUNG
   // the same network as SCL:
   IF NOT #SYS_SIGNALS._False THEN
       #licInfo.LICENCE_TYPE := 'MIT LICENSE';
       #licInfo.COPYRIGHT := '2020 Michael Gledhill';
   END_IF;
END_REGION
END_FUNCTION

FUNCTION "FC18001_StdSubScaleAI" : Void   // FC18001, LAD
TITLE = Standard Module [SUBROUTINE] — Analog Input Scale
{ S7_Optimized_Access := 'TRUE' }
AUTHOR : M_Gledhill
FAMILY : Subroutine
NAME : StdSubScaleAI
VERSION : 2.0
// PRACTICAL SERIES AUTOMATION LIBRARY (PAL)   —   COPYRIGHT 2020 – M. GLEDHILL (MIT LICENCE)
//                   ———— ◆ ————
// FULL ONLINE DOCUMENTATION IS AVAILABLE AT: https://practicalseries.com/2001-pal/index.html
// stored: AutoNumber false, IsIECCheckEnabled true, SetENOAutomatically false, UDAEnableTagReadback false
   VAR_INPUT
      SYS_SIGNALS : "UT21000_Dy_SysSignals";   // The system logic and timing signals for parametric access
      RAW_ANALOG : Int;   // Analogue Input (IW)
      RAW_MIN : Int;   // Minimum Valve of the Raw Analogue Input
      RAW_MAX : Int;   // Maximum Valve of the Raw Analogue Input
      SCALE_MIN : Real;   // Minimum value of the scaled output (engineering units)
      SCALE_MAX : Real;   // Maximum value of the scaled output(engineering units)
      OOR_PERCENT : Real;   // Out of range tolerance as a percentage of raw range (RAW_MAX - RAW_MIN)
   END_VAR
   VAR_OUTPUT
      SCALE_VALUE : Real;   // Scaled Output (as a Floating Point value)
      OVER_RANGE : Bool;   // Signal Fault - Over range
      UNDER_RANGE : Bool;   // Signal Fault - Under range
      OUT_OF_RANGE : Bool;   // Signal Fault - Out of Range (either over or under)
   END_VAR
   VAR_TEMP
      revInfo : "UT01000_St_SysRevision";   // Revision information for this block
      licInfo : "UT01001_St_SysLicence";   // Licence information for this block
      calPart1 : Real;   // Scale value calculation part 1 (RAW_ANALOG − RAW_MIN)
      calPart2 : Real;   // Scale value calculation part 2 (SCALE_MAX − SCALE_MIN)
      calPart3 : Real;   // Scale value calculation part 1 (RAW_MAX − RAW_MIN)
      calAbsOOR : Real;   // Calculated OOR absolute value in terms of the RAW_VALUE
      calOverRange : Real;   // Calculated over range limit (in raw units)
      calUnderRange : Real;   // Calculated under range limit (in raw units)
      wrkOORPercent : Real;   // Working out of range percentage
      wrkConfigError : Bool;   // Working configuration error exists
      wrkReal : Real;   // Working storage (real)
   END_VAR
BEGIN

REGION Network 1: Block description
   // ▄▄▄▄▄▄▄▄▄▄▄▄▄▄▄▄▄▄▄▄▄▄▄▄▄▄▄▄▄▄▄▄▄  ＳＴＡＮＤＡＲＤ  ▄▄ 
   // 
   // 
   // TITLE:    SUBROUTINE — ANALOG INPUT SCALE
   // 
   // 
   // ▀▀▀▀▀▀▀▀▀▀▀▀▀▀▀▀▀▀▀▀▀▀▀▀▀▀▀▀▀▀▀▀▀▀▀▀▀▀▀▀▀▀▀▀ 
   // 
   // ┌──────────────────────────────────────────┐
   // │                                          │
   // │          FC18001 — SOFTWARE MODULE DESIGN SPECIFICATION (SMDS)            │
   // │                                          │
   // │      The PDF version of the SMDS for this module is available online here:        │
   // │              http://psop.uk/pal-smds-fc18001-p              │
   // │                                          │
   // │      It is also available as part of the Project User Defined Documentation,      │
   // │      it can be accessed by selecting this module in the Project Tree          │
   // │      (on the left) and pressing SHIFT+F1                        │
   // │                                          │
   // └─────────────────────────────────────── ʷᴵᴰ⁻ᵇᵈᵖ ┘
   // 
   // FC18001_StdSubScaleAI is a subroutine block that is used to scale the integer signal from an 
   // analog instrument, in the form of an input word (IW).
   // 
   // The resultant scaled value is a real (floating point) number that matches the calibrated range 
   // of the instrument.
   // 
   // The block monitors the instrument to see if the scaled value is out-of-range, the following three 
   // fault signals are generated:
   // 
   //    •   Over-range (signal is more than a specified percentage above the calibrated 
   //      range of the instrument
   // 
   //    •   Under-range (signal is more than a specified percentage below the calibrated 
   //      range of the instrument
   // 
   //    •   Common out-of-range, either the over-range or under-range fault is active
   // 
   // This is a subroutine block.
   // 
   // 
   // 
   // ▄▄▄▄▄▄▄▄▄▄▄▄▄▄▄▄▄▄▄▄▄▄▄▄▄▄▄▄▄▄▄▄▄▄▄▄▄▄▄▄▄▄▄▄
   // 1.     BLOCK TECHNICAL SUMMARY
   // 
   // 
   //  ――――――――――――――――――――――――――――――――――――――――――
   //  NOMENCLATURE & ADDRESSING
   //  ――――――――――――――――――――――――――――――――――――――――――
   //  BLOCK TITLE         Analog Input Scale
   //  BLOCK FUNCTION GROUP    Subroutine
   //  BLOCK ADDRESS       FC18001
   //  BLOCK SYMBOL        FC18001_StdSubScaleAI
   //  BLOCK USER ID         StdSubScaleAI
   // 
   //  ――――――――――――――――――――――――――――――――――――――――――
   //  BLOCK TYPE & USAGE
   //  ――――――――――――――――――――――――――――――――――――――――――
   //  BLOCK TYPE         Function (FC)
   //  BLOCK NUMBER        18001
   //  LANGUAGE           LAD
   //  OPTIMISED ACCESS     Yes
   //  PAL USAGE TYPE       Standard block
   // 
   //  ――――――――――――――――――――――――――――――――――――――――――
   //  METRICS
   //  ――――――――――――――――――――――――――――――――――――――――――
   //  EXECUTION TIME       23.9 μs¹
   //  LOAD MEMORY       28.3 kB
   //  WORK MEMORY           0.6 kB  
   //  ――――――――――――――――――――――――――――――――――――――――――
   //                ¹ Measured on: CPU-1515-2PN (order no. 6ES7512-2AM02-0AB0) 
   //                             http://psop.uk/pal-ds-cpu1515
   // 
   // 
   // 
   // ▂▂▂▂▂▂▂▂▂▂▂▂▂▂▂▂▂▂▂▂▂▂▂▂▂▂▂▂▂▂▂▂▂▂▂▂▂▂▂▂▂▂▂▂
   // 1.1      Additional document references
   // 
   // 
   // Only those documents specified in OB1 (section DOCUMENT REFERENCES) are listed within this 
   // block. There are no additional document references.
   // 
   //                ━━━   ⬙⬙⬙⬙⬙⬙   ━━━
   // 
   // 
   // 
   // ▄▄▄▄▄▄▄▄▄▄▄▄▄▄▄▄▄▄▄▄▄▄▄▄▄▄▄▄▄▄▄▄▄▄▄▄▄▄▄▄▄▄▄▄
   // 2.     FUNCTIONAL DESCRIPTION
   // 
   // 
   // This is a subroutine block that is used to convert the raw integer signal from an analog 
   // instrument (in the form of an input word, IW), into a scaled, floating point (real) number that 
   // reflects the calibrated reading of the instrument in question.
   // 
   // For example, if a flow meter with a calibrated range of -100 l/s to +100 l/s provided a 4-20 mA 
   // signal to the PLC, then 4 mA would represent -100 l/s and 20 mA would represent +100 l/s.
   // 
   // A typical 4-20 mA analog input signal returns raw value of 0 at 4 mA and 27648 at 20 mA.
   // 
   // The block would return scaled values as follows (it would also return every value in between; five 
   // typical values have been shown):
   // 
   // 
   //  ――――――――――――――――――――――――――――――――――――――――――
   //  RAW_SIGNAL          RAW INTEGER VALUE        RETURNED SCALE VALUE
   //  ――――――――――――――――――――――――――――――――――――――――――
   //     4 mA                      0             -100 l/s
   //     8 mA               6912                   -50 l/s
   //   12 mA             13824                   0 l/s
   //   16 mA             20736              +50 l/s
   //   20 mA             27648            +100 l/s
   //  ――――――――――――――――――――――――――――――――――――――――――
   // 
   // 
   // The range of the raw instrument signal is specified by the parameters RAW_MIN (the lowest 
   // value the instrument will read in its calibrated normal range) and RAW_MAX (the highest 
   // value the instrument will read in its normal calibrated range).
   // 
   // The scaled value has two equivalent parameters: SCALE_MIN (the lowest value of the 
   // instrument in its calibrated range in engineering units) and SCALE_MAX (the highest value 
   // of the instrument in its calibrated range in engineering units).
   // 
   // In the previous example, the parameters would be:
   // 
   // 
   //  ――――――――――――――――――――――――――――――――――――――――――
   //  RAW_MIN       RAW_MAX      SCALE_MIN       SCALE_MAX
   //  ――――――――――――――――――――――――――――――――――――――――――
   //       0         27648            -100.0         +100.0
   //  ――――――――――――――――――――――――――――――――――――――――――
   // 
   // 
   // The actual raw instrument value is passed to the block as parameter RAW_ANALOG, this is of data 
   // type int. The resultant scaled signal is passed from the block as the parameter SCALE_VALUE
   // of type real.
   // 
   // The block generates three fault signals, these indicate if the instrument is reading above its 
   // normal, calibrated range by a specified amount, or if it is reading below its calibrated range by a 
   // similar amount (these are, respectively, the OVER_RANGE and UNDER_RANGE parameters). The 
   // third fault signal (OUT_OF_RANGE) is simply a common signal that is activated if either of the 
   // other two is active.
   // 
   // The level at which the instrument is considered to be either over-range or under-range 
   // (out-of-range), is set as a percentage of the raw instrument range and is specified in the 
   // OOR_PERCENT parameter (this is limited to a range of 0.0 to 10.0% of the raw instrument 
   // range). 
   // 
   // Note:    The instrument must have a linear response across its calibrated range.
   // 
   // 
   // 
   // ▄▄▄▄▄▄▄▄▄▄▄▄▄▄▄▄▄▄▄▄▄▄▄▄▄▄▄▄▄▄▄▄▄▄▄▄▄▄▄▄▄▄▄▄
   // 3.     DETAILED BLOCK DESCRIPTION
   // 
   // 
   // This block, FC18001_StdSubAnalogScaleAI is a subroutine block that can be called from other 
   // blocks within the PAL. It is designed to provide a linear conversion of a raw analog input signal 
   // (in integer format) to a scaled value that represents the calibrated range of the instrument as a 
   // real (floating point) value in engineering units.
   // 
   // It has the following formal parameters:
   // 
   // 
   //  ――――――――――――――――――――――――――――――――――――――――――
   //  PARAM         FUNCTION                    TYPE      IN-OUT 
   //  ――――――――――――――――――――――――――――――――――――――――――
   //  SYS_SIGNALS      The system logic and timing signals for       UT21000    In
   //           parametric access
   // 
   //  RAW_ANALOG      Analog input signal (IW) to be scaled. This is       Int      In
   //           the raw value returned from the AI card
   // 
   //  RAW_MIN     Minimum value of the analog input range        Int      In
   //           (see Table 3.1 to Table 3.3 for typical values)
   // 
   //  RAW_MAX       Maximum value of the analog input range        Int      In
   //           (see Table 3.1 to Table 3.3 for typical values)
   // 
   //  SCALE_MIN    Calibrated lower value of the instrument       Real      In
   //           range in engineering units
   // 
   //  SCALE_MAX      Calibrated upper value of the instrument      Real      In
   //           range in engineering units
   // 
   //  OOR_PERCENT     Out of range tolerance as a percentage of    Real      In
   //           the raw range (RAW_MAX − RAW_MIN), the value 
   //           is limited to the range 0.001% to 10.0%
   // 
   //  SCALE_VALUE     The scaled output value of the instrument in      Real      Out
   //           engineering units
   // 
   //  OVER_RANGE      Indicates the instrument is above its        Bool      Out
   //           calibrated range by more than the tolerance
   //           value (OOR_PERCENT)
   // 
   //  UNDER_RANGE    Indicates the instrument is below its        Bool      Out
   //           calibrated range by more than the tolerance 
   //           value (OOR_PERCENT)
   // 
   //  OUT_OF_RANGE     Indicates the instrument is outside of its       Bool      Out
   //           calibrated range by more than the tolerance 
   //           value (OOR_PERCENT), either over or 
   //           under range
   //  ――――――――――――――――――――――――――――――――――――――――――
   //  Note:   If a configuration error is present (see § 3.2.1) the three out of range parameters 
   //      will be activated (set true) and the SCALE_VALUE signal will be set to zero 
   //      irrespective of the RAW_ANALOG value.
   // 
   // 
   // 
   // ▂▂▂▂▂▂▂▂▂▂▂▂▂▂▂▂▂▂▂▂▂▂▂▂▂▂▂▂▂▂▂▂▂▂▂▂▂▂▂▂▂▂▂▂
   // 3.1     Raw signal, typical ranges
   // 
   // 
   // The raw (unscaled) instrument value is the value returned from the analog input card. This 
   // typically is ranged according to the type of signal being read (voltage, current, RTD &c.). 
   // 
   // The raw instrument value (the value provided by the analog input card) is passed to the block 
   // as parameter RAW_ANALOG. The associated range of the signal is given in parameters RAW_MIN 
   // and RAW_MAX.
   // 
   // The following are the typical signal ranges for the most common types of signals:
   // 
   // 
   //  ――――――――――――――――――――――――――――――――――――――――――
   //             LOWER LIMIT     EQUIVALENT   UPPER LIMIT     EQUIVALENT
   //  SIGNAL TYPE      (RAW_MIN)          TO      (RAW_MAX)         TO
   //  ――――――――――――――――――――――――――――――――――――――――――
   //  -10 V to 10 V         -27648      -10 V          27648        +10 V
   //  -5 V to 5 V       -27648        -5 V          27648       +5 V
   //  -2.5 V to 2.5 V       -27648        -2.5 V          27648       +2.5 V
   //  -1 V to 1 V       -27648        -1 V          27648       +1 V
   //  -500 mV to 500 mV      -27648       -500 mV      27648      +500 mV
   //  -250 mV to 250 mV      -27648       -250 mV      27648      +250 mV
   //  -80 mV to 80 mV       -27648      -80 mV      27648        +80 mV
   //  -50 mV to 50 mV    -27648      -50 mV      27648        +50 mV
   //  1 V to 5 V          0       +1 V          27648       +5 V
   //  ――――――――――――――――――――――――――――――――――――――――――
   //  Table 3.1  Input ranges for typical instrument types (voltage)
   // 
   // 
   // 
   //  ――――――――――――――――――――――――――――――――――――――――――
   //             LOWER LIMIT     EQUIVALENT   UPPER LIMIT     EQUIVALENT
   //  SIGNAL TYPE      (RAW_MIN)          TO      (RAW_MAX)         TO
   //  ――――――――――――――――――――――――――――――――――――――――――
   //  -500 mV to 500 mV   -27648       -500 mV      27648      +500 mV
   //  -20 mA to 20 mA       -27648      -20 mA      27648        +20 mA
   //  0 mA to 20 mA         0         0 mA      27648        +20 mA
   //  4 mA to 20 mA         0         4 mA      27648        +20 mA
   //  ――――――――――――――――――――――――――――――――――――――――――
   //  Table 3.2  Input ranges for typical instrument types (current)
   // 
   // 
   // 
   //  ――――――――――――――――――――――――――――――――――――――――――
   //             LOWER LIMIT     EQUIVALENT   UPPER LIMIT     EQUIVALENT
   //  SIGNAL TYPE      (RAW_MIN)          TO      (RAW_MAX)         TO
   //  ――――――――――――――――――――――――――――――――――――――――――
   //  -500 mV to 500 mV   -27648       -500 mV      27648      +500 mV
   //  RTD 150 Ω            0         0 Ω         27648        150 Ω
   //  RTD 300 Ω            0         0 Ω         27648        300 Ω
   //  RTD 600 Ω            0         0 Ω         27648        600 Ω
   //  RTD 6000 Ω         0         0 Ω         27648      6000 Ω
   //  PT x00           -2000        200.0°C        8500        850.0°C
   //  Ni x00          -600       60.0°C          250        250.0°C
   //  Type B thermocouple     -2100       -210.0°C        12000      1200.0°C
   //  Type K thermocouple     -2700       -270.0°C        13720      1372.0°C
   //  Type N thermocouple    -2700       -210.0°C        13000      1300.0°C
   //  Type R/S thermocouple    -500      -50.0°C        17690      1769.0°C
   //  Type T thermocouple     -2700       -270.0°C        4000        400.0°C
   //  ――――――――――――――――――――――――――――――――――――――――――
   //  Table 3.3  Input ranges for typical instrument types (resistance thermometers 
   //           and thermocouples)
   // 
   // 
   // The RAW_MIN and the RAW_MAX values in the above tables are the numerical values for the 
   // instrument range; the appropriate values must be entered as parameters passed to the block:
   // 
   // 
   //  ――――――――――――――――――――――――――――――――――――――――――
   //  PARAM         FUNCTION                  TYPE      IN-OUT 
   //  ――――――――――――――――――――――――――――――――――――――――――
   //  RAW_MIN     Minimum value of the analog input range      Int      In
   // 
   //  RAW_MAX       Maximum value of the analog input range      Int      In
   //  ――――――――――――――――――――――――――――――――――――――――――
   // 
   //  
   // 
   // ▂▂▂▂▂▂▂▂▂▂▂▂▂▂▂▂▂▂▂▂▂▂▂▂▂▂▂▂▂▂▂▂▂▂▂▂▂▂▂▂▂▂▂▂
   // 3.2     Calculating the scaled value
   // 
   // 
   // The scaled signal is passed from the block as parameter SCALE_VALUE and this in turn is ranged 
   // between the SCALE_MIN and SCALE_MAX parameters. SCALE_MIN is the lowest calibrated 
   // reading of the instrument in engineering units and SCALE_MAX being the upper calibrated 
   // reading of the instruments in engineering units.
   // 
   // The formula used to calculate the scaled value (SCALE_VALUE) is:
   // 
   // ┌──────────────────────────────────────────┐
   // │                                    (RAW_ANALOG ─ RAW_MIN) ╳ (SCALE_MAX ─ SCALE_MIN)          │
   // │ SCALE_VALUE =  ――――――――――――――――――――――――――  ┼ SCALE_MIN   │
   // │                                    (RAW_MAX ─ RAW_MIN)                  │
   // └─────────────────────────────────────  (3.1)  ──┘
   // 
   // The three parameters: SCALE_VALUE, SCALE_MIN and SCALE_MAX are all floating-point numbers 
   // (real data type).
   // 
   // Note:    It is assumed that the instrument must have a linear response across its calibrated 
   //      range (as shown below).
   // 
   // 
   //       SCALE_VALUE
   //        ↑                    ⋰
   //    SCALE_MAX__│______________________________________⋰
   //        │                  ╱|
   //        │                 ╱ |
   //        │                ╱  |
   //        │               ╱   |
   //        │              ╱    |
   //        │             ╱     |
   //        │            ╱      |
   //    SCALE_VALUE│<- - - - - - - - - - - - - - - - - - - - - ╱       |
   //        │          ╱ ⌃           |
   //        │         ╱ ╎       |
   //        │        ╱  ╎       |
   //        │       ╱   ╎       |   
   //        │      ╱    ╎       |
   //        │     ╱     ╎       |
   //        │    ╱         ╎          |
   //  SCALE_MIN__│______╱          ╎          |
   //        │  ⋰|           ╎          |
   //        │ ⋰ |           ╎          |
   //        ┼─────────────────────────→ RAW_ANALOG
   //              |           ╎           |
   //          RAW_MIN     RAW_ANALOG    RAW_MAX
   // 
   //        Linear relationship between RAW_ANALOG and SCALE_VALUE
   // 
   // 
   // 
   // ▁▁▁▁▁▁▁▁▁▁▁▁▁▁▁▁▁▁▁▁▁▁▁▁▁▁▁▁▁▁▁▁▁▁▁▁▁▁▁▁▁▁▁▁
   // 3.2.1     Configuration errors
   // 
   // 
   // The block requires that both the RAW_MAX/MIN and SCALE_MAX/MIN signals conform to certain 
   // rules:
   // 
   //    1.  RAW_MIN must be less than, and not equal to RAW_MAX
   //    2.  SCALE_MIN must be less than, and not equal to SCALE_MAX
   // 
   // Should either of these conditions not be met, the three out of range parameters (see § 3.3.1) will 
   // be activated (set true) 
   // 
   //      OVER_RANGE
   //      UNDER_RANGE
   //      OUT_OF_RANGE
   // 
   // The SCALE_VALUE signal will be set to zero irrespective of the RAW_ANALOG value.
   // 
   // Note:    This avoids the potential for a divide by zero error, if the RANGE_RAW_MIN and 
   //      RANGE_RAW_MAX are exactly equal, the calculation of the actual_Value in 
   //      equation (3.1) would result in a divide by zero error. 
   // 
   // 
   // 
   // ▂▂▂▂▂▂▂▂▂▂▂▂▂▂▂▂▂▂▂▂▂▂▂▂▂▂▂▂▂▂▂▂▂▂▂▂▂▂▂▂▂▂▂▂
   // 3.3     Out of range signals
   // 
   // 
   // If the RAW_ANALOG signal is outside the RAW_MIN to RAW_MAX range, SCALE_VALUE will still be 
   // calculated correctly; however, an appropriate, OVER_RANGE or UNDER_RANGE signal will be 
   // generated to indicate that the SCALE_VALUE signal is outside the calibrated range of the 
   // instrument and is potentially no longer accurate.
   // 
   // Some tolerance is permitted before the OVER_RANGE and UNDER_RANGE signals are activated 
   // (this is to prevent nuisance alarms — most instruments are tolerant of slight over and under 
   // shoot readings).
   // 
   // The tolerance applied to the out of range signals is a percentage of the raw range of the 
   // instrument (the raw range being RAW_MAX − RAW_MIN). 
   // 
   // The tolerance to be applied is given in the parameter OOR_PERCENT, this is a real (floating point) 
   // number in the range 0.0-10.0%.
   // 
   // If the tolerance for the instrument is not known, a generic value of 2.5% should be used.
   // 
   // The out of range tolerance absolute value (in terms of the RAW_ANALOG rather than as a
   // percentage) is calculated as:
   // 
   // ┌─────────────────────────────┐
   // │                                 (RAW_MAX ─ RAW_MIN) ╳ OOR_PERCENT    │
   // │ calAbsOOR =  ―――――――――――――――――――     │
   // │                  100          │
   // └────────────────────────  (3.2)  ──┘
   // 
   // Thus, if RAW_MIN is 0, RAW_MAX is 27648 and an OOR_PERCENT of 2.5% is selected, the 
   // absolute out of range value (calAbsOOR in the above equation) has a calculated value 
   // of 691. 
   // 
   // In this example, the OVER_RANGE signal would activate when the RAW_ANALOG exceeded a 
   // value of RAW_MAX + 691 (or 28,339). The UNDER_RANGE signal would activate when the 
   // RAW_ANALOG fell below a value of RAW_MIN ─ 691 (or −691).
   // 
   // The OOR_PERCENT is applied directly to the RAW_ANALOG signal, however, because the 
   // instrument is considered to be linear, the same calculation can also be applied directly to 
   // the SCALE_VALUE. In the above example, if the instrument were to span the range of 
   // −100 l/s to +100 l/s (i.e. SCALE_MIN = −100 SCALE_MAX = +100) then the scaled range of the 
   // instrument is 200 l/s (SCALE_MAX ─ SCALE_MIN) and the absolute out of range value would 
   // be 2.5% of the scaled range (or 5 l/s). thus, the OVER_RANGE signal would activate above 105 l/s 
   // and the UNDER_RANGE signal would activate below −105 l/s.
   // 
   // The OOR_PERCENT must be in the range 0.0 to 10.0; If it is outside this range, it 
   // is fixed at either the upper or lower limit.
   // 
   // 
   // 
   // ▁▁▁▁▁▁▁▁▁▁▁▁▁▁▁▁▁▁▁▁▁▁▁▁▁▁▁▁▁▁▁▁▁▁▁▁▁▁▁▁▁▁▁▁
   // 3.3.1     Common out of range signal
   // 
   // 
   // There is a third out of range signal: OUT_OF_RANGE, this signal is a common signal that just 
   // indicates the instrument is out of its calibrated range (it does not specify whether it is over or 
   // under range). 
   // 
   // It is activated if either the OVER_RANGE or UNDER_RANGE signal is active.
   // 
   // Note:    If a configuration error exists, see § 3.2.1, all three out of range signals (OVER_RANGE, 
   //      UNDER_RANGE and OUT_OF_RANGE) will be activated irrespective of the 
   //      RAW_ANALOG value
   // 
   //                ━━━   ⬙⬙⬙⬙⬙⬙   ━━━
   // 
   // 
   // 
   // ▄▄▄▄▄▄▄▄▄▄▄▄▄▄▄▄▄▄▄▄▄▄▄▄▄▄▄▄▄▄▄▄▄▄▄▄▄▄▄▄▄▄▄▄
   // 4.     Supervisory system interface
   // 
   // 
   // FC18001 is a Subroutine block used to scale an analog input. 
   // 
   // It does not have a supervisory system interface.
   // 
   // 
   //                ━━━   ⬙⬙⬙⬙⬙⬙   ━━━
   // 
   // 
   // 
   // ▄▄▄▄▄▄▄▄▄▄▄▄▄▄▄▄▄▄▄▄▄▄▄▄▄▄▄▄▄▄▄▄▄▄▄▄▄▄▄▄▄▄▄▄
   // 5.     PARAMETERS
   // 
   // 
   // The following parameters are associated with the block:
   // 
   //  
   //  ――――――――――――――――――――――――――――――――――――――――――
   //  PARAM         FUNCTION                    TYPE      IN-OUT 
   //  ――――――――――――――――――――――――――――――――――――――――――
   //  SYS_SIGNALS      The system logic and timing signals for       UT21000    In
   //           parametric access
   // 
   //  RAW_ANALOG      Analog input signal (IW) to be scaled. This is       Int      In
   //           the raw value returned from the AI card
   // 
   //  RAW_MIN     Minimum value of the analog input range        Int      In
   //           (see Table 3.1 to Table 3.3 for typical values)
   // 
   //  RAW_MAX       Maximum value of the analog input range        Int      In
   //           (see Table 3.1 to Table 3.3 for typical values)
   // 
   //  SCALE_MIN    Calibrated lower value of the instrument       Real      In
   //           range in engineering units
   // 
   //  SCALE_MAX      Calibrated upper value of the instrument      Real      In
   //           range in engineering units
   // 
   //  OOR_PERCENT     Out of range tolerance as a percentage of    Real      In
   //           the raw range (RAW_MAX − RAW_MIN), the value 
   //           is limited to the range 0.001% to 10.0%
   // 
   //  SCALE_VALUE     The scaled output value of the instrument in      Real      Out
   //           engineering units
   // 
   //  OVER_RANGE      Indicates the instrument is above its        Bool      Out
   //           calibrated range by more than the tolerance
   //           value (OOR_PERCENT)
   // 
   //  UNDER_RANGE    Indicates the instrument is below its        Bool      Out
   //           calibrated range by more than the tolerance 
   //           value (OOR_PERCENT)
   // 
   //  OUT_OF_RANGE     Indicates the instrument is outside of its       Bool      Out
   //           calibrated range by more than the tolerance 
   //           value (OOR_PERCENT), either over or 
   //           under range
   //  ――――――――――――――――――――――――――――――――――――――――――
   //  Note:   If a configuration error is present (see § 3.2.1) the three out of range parameters 
   //      will be activated (set true) and the SCALE_VALUE signal will be set to zero 
   //      irrespective of the RAW_ANALOG value
   // 
   //                ━━━   ⬙⬙⬙⬙⬙⬙   ━━━
   // 
   // 
   // 
   // ▄▄▄▄▄▄▄▄▄▄▄▄▄▄▄▄▄▄▄▄▄▄▄▄▄▄▄▄▄▄▄▄▄▄▄▄▄▄▄▄▄▄▄▄
   // 6.     DATA STRUCTURES AND USAGE
   // 
   // 
   // The block has the following associated data structure:
   // 
   // 
   //  ――――――――――――――――――――――――――――――――――――――――――
   //  DATA STRUCTURE             DESCRIPTION
   //  ――――――――――――――――――――――――――――――――――――――――――
   //  UT01000_St_SysRevision          Revision information for this block    See FC01001
   //  UT01001_St_SysLicence           Licence information for this block  See FC01001
   //  UT21000_Dy_SysSignals           System signals for logic and timing  See FC01001
   //  ――――――――――――――――――――――――――――――――――――――――――
   // 
   //                ━━━   ⬙⬙⬙⬙⬙⬙   ━━━
   // 
   // 
   // 
   // ▄▄▄▄▄▄▄▄▄▄▄▄▄▄▄▄▄▄▄▄▄▄▄▄▄▄▄▄▄▄▄▄▄▄▄▄▄▄▄▄▄▄▄▄
   // 7.     CONSTANTS AND TEMPORARY (LOCAL) DATA
   // 
   // 
   // 
   // ▂▂▂▂▂▂▂▂▂▂▂▂▂▂▂▂▂▂▂▂▂▂▂▂▂▂▂▂▂▂▂▂▂▂▂▂▂▂▂▂▂▂▂▂
   // 7.1     Constants
   // 
   // 
   // No constants are used in this block.
   // 
   // 
   // 
   // ▂▂▂▂▂▂▂▂▂▂▂▂▂▂▂▂▂▂▂▂▂▂▂▂▂▂▂▂▂▂▂▂▂▂▂▂▂▂▂▂▂▂▂▂
   // 7.2     Temporary (local) data
   // 
   // 
   // The following temporary data is used:
   // 
   //  ――――――――――――――――――――――――――――――――――――――――――
   //  SIGNAL NAME          FUNCTION                  TYPE
   //  ――――――――――――――――――――――――――――――――――――――――――
   //  revInfo             Revision information for the block         UT01000
   //  licInfo           Licensing information for the block      UT01001
   //  calPart1             Scale value part 1 (RAW_ANALOG − RAW_MIN)    Real
   //  calPart2             Scale value part 2 (SCALE_MAX − SCALE_MIN)   Real
   //  calPart3             Scale value part 3 (RAW_MAX − RAW_MIN)     Real
   //  calAbsOOR           Calculated OOR absolute value          Real
   //  calOverRange         Calculated over range limit (in raw units)    Real
   //  calUnderRange         Calculated under range limit (in raw units)     Real
   //  wrkOORPercent         Working out of range percentage       Real
   //  wrkConfigError        Working configuration error exists         Bool
   //  wrkReal           Working storage (Real)             Real
   //  ―――――――――――――――――――――――――――――――――――――――――
   // 
   //                ━━━   ⬙⬙⬙⬙⬙⬙   ━━━
   // 
   // 
   // 
   // ▄▄▄▄▄▄▄▄▄▄▄▄▄▄▄▄▄▄▄▄▄▄▄▄▄▄▄▄▄▄▄▄▄▄▄▄▄▄▄▄▄▄▄▄
   // 8.     BLOCK CALLS AND ASSOCIATIONS
   // 
   // 
   // This section details any blocks which may be called from within this software module (subroutine 
   // functions for example), any partner blocks with which it may be associated (for example a 
   // receive module that is partner with a transmit module &c.). It lists any system functions which 
   // may be called (e.g. reading the real time clock) and any system data types that may be used.
   // 
   // Finally, it lists any special calling requirements for the block (for example, must be called from 
   // within a cyclic interrupt organisation block) and if the block is using “optimised access” (this is 
   // the default arrangement).
   // 
   // 
   // 
   // ▂▂▂▂▂▂▂▂▂▂▂▂▂▂▂▂▂▂▂▂▂▂▂▂▂▂▂▂▂▂▂▂▂▂▂▂▂▂▂▂▂▂▂▂
   // 8.1     Block calls from within this module
   // 
   // 
   // There are no PAL block calls from within this block.
   // 
   // 
   // 
   // ▂▂▂▂▂▂▂▂▂▂▂▂▂▂▂▂▂▂▂▂▂▂▂▂▂▂▂▂▂▂▂▂▂▂▂▂▂▂▂▂▂▂▂▂
   // 8.2     Blocks associated with this module
   // 
   // 
   // This is a stand-alone block and is not associated with any other blocks.
   // 
   // 
   // 
   // ▂▂▂▂▂▂▂▂▂▂▂▂▂▂▂▂▂▂▂▂▂▂▂▂▂▂▂▂▂▂▂▂▂▂▂▂▂▂▂▂▂▂▂▂
   // 8.3     System block calls and system data types
   // 
   // There are no system block calls
   // 
   // 
   // 
   // ▂▂▂▂▂▂▂▂▂▂▂▂▂▂▂▂▂▂▂▂▂▂▂▂▂▂▂▂▂▂▂▂▂▂▂▂▂▂▂▂▂▂▂▂
   // 8.4     Special properties and requirements
   // 
   // 
   // 
   // ▁▁▁▁▁▁▁▁▁▁▁▁▁▁▁▁▁▁▁▁▁▁▁▁▁▁▁▁▁▁▁▁▁▁▁▁▁▁▁▁▁▁▁▁
   // 8.4.1     Block optimisation, IEC compatibility and library conformance
   // 
   // 
   //    •   Block optimisation is ACTIVE for this block.
   // 
   //    •   The block has been checked for IEC compatibility and is compliant.
   // 
   //    •   The block is compatible with all IEC library-conformance module constraints
   // 
   // 
   // 
   // ▁▁▁▁▁▁▁▁▁▁▁▁▁▁▁▁▁▁▁▁▁▁▁▁▁▁▁▁▁▁▁▁▁▁▁▁▁▁▁▁▁▁▁▁
   // 8.4.2     Calling requirements
   // 
   // 
   // There are no special calling requirements for this block.
   // 
   //                ━━━   ⬙⬙⬙⬙⬙⬙   ━━━
   // 
   // 
   // 
   // ▄▄▄▄▄▄▄▄▄▄▄▄▄▄▄▄▄▄▄▄▄▄▄▄▄▄▄▄▄▄▄▄▄▄▄▄▄▄▄▄▄▄▄▄
   // 9.     EXAMPLE USAGE
   // 
   // 
   // The following shows a typical deployment of FC18001:
   // 
   //                ┌─────────────
   //  ──────────────┤ FC18001
   //                ├───────────
   //                │
   //        #SYS_SIGNALS ─┤ SYS_SIGNALS
   //                │
   //        #RAW_ANALOG ─┤ RAW_ANALOG
   //                │
   //                 0 ─┤ RAW_MIN
   //                │
   //              27648 ─┤ RAW_MAX       SCALE_VALUE├─ #VALUE
   //                │                 │
   //              -100.0 ─┤ SCALE_MIN        UNDER_RANGE ├─ #ALM_OOR
   //                │                 │
   //               100.0 ─┤ SCALE_MAX       OVER_RANGE├─ #ALM_OVER_R
   //                │                 │
   //                    2.5 ─┤ OOR_PERCENT       OUT_OF_RANGE├─ #ALM_UNDER_R  
   //                │                 │
   //                                  │
   //                     ─────────────┘
   // 
   // 
   //                ━━━   ⬙⬙⬙⬙⬙⬙   ━━━
   // 
   // 
   // 
   // ▄▄▄▄▄▄▄▄▄▄▄▄▄▄▄▄▄▄▄▄▄▄▄▄▄▄▄▄▄▄▄▄▄▄▄▄▄▄▄▄▄▄▄▄
   // 10.     TEST AND VERIFICATION PATH
   // 
   // 
   // The following diagram shows the full test and verification path for the formal release of each 
   // version of the software module. See the Test Plan [Ref. 003] for full details, available here:
   //         http://psop.uk/pal-tp-p
   // 
   // 
   //         FC18001-T001         FC18001-T002
   // 
   //     Test version: 000.801     Test version: 001.801
   //  Released version: 001.000     Released version: 002.000
   // Released commit: D0007    Released commit: D0011
   // 
   //        SCR      SMT              SCV     
   // ＿＿＿＿＿＿┌┐＿＿ ▛▜ ＿＿＿＿＿＿＿＿＿＿＿＿╓╖＿＿
   //       └┘   ▙▟             ╙╜  
   // Initial test           Comments standardised
   // 
   // Initial test to release the      Comments updated & 
   // module following the      minor typographical 
   // development stage.       corrections
   // Full SMT              SCV only
   // 
   // 
   // Where:
   // ――――――――――――――――――――――――――――――――――――――――――――
   //  SCR    Source Code Review      A visual inspection of the software to ensure it has been written  
   // ┌┐             to the correct standards, uses the correct structures within the
   // └┘             software and is generally suitable for deployment.               
   // 
   //  SMT Software Module Test    A full and detailed test of an individual software module in
   //   ▛▜              isolation; such testing requires that all branches of the 
   //   ▙▟              software are tested. 
   // 
   //                It tests all the interfaces to the module, any data recorded or 
   //                stored by the module, all error and exception handling functions 
   //                and tests all timed and interrupt driven operations.
   // 
   //  SCV Software Compatibility     A mechanism for verifying that no executable code software 
   // ╓╖    Verification          changes have been made to a module following changes to
   // ╙╜             comment fields.
   // 
   //                Allows typographical errors &c. to be corrected without forcing 
   //                a full SMT on a module that has not functionally changed.
   // ――――――――――――――――――――――――――――――――――――――――――――
   // 
   // An SCV can only be performed on a module that has at some point previously, successfully 
   // completed both an SCR and SMT. Where an SCV is implemented, it replaces the requirement for 
   // both the SCR and the SMT for the test iteration in question.
   // 
   //                ━━━   ⬙⬙⬙⬙⬙⬙   ━━━
   // 
   // 
   // ██████████████ █ █ █ █  END   █ █ █ █ ██████████████
END_REGION

REGION Network 2: Current revision and modification history
   // ▄▄▄▄▄▄▄▄▄▄▄▄▄▄▄▄▄▄▄▄▄▄▄▄▄▄▄▄▄▄▄▄▄▄▄▄▄▄▄▄▄▄▄▄
   // MODIFICATION HISTORY
   // 
   // 
   // The revision data shown here, in the network comments, contains additional information 
   // reflecting the software development workflow under the version control system (VCS) employed 
   // to track all software changes.
   // 
   // The VCS in use is the Git Source Code Management system in conjunction with the GitHub online 
   // hosting system. The software in its entirety is available in the GitHub remote repository:
   // 
   //      https://github.com/practicalseries/PS2001-pal-software
   // 
   // The repository is public and can be freely copied (forked in GitHub terminology) and used 
   // under the MIT licence. 
   // 
   // The MIT licence is reproduced in full in the last network of this software module.
   // 
   // 
   //  ―――――――――――――――――――――――――――――――――――――――――――
   //  DATE       REVISION             MASTER BRANCH     DEV
   //          (nnn.amm)   COMMIT TAG    (Base ---> Merge)    BRANCH   Author
   //  ———————————————————————————————————————————
   //  2022.04.16    002.000   D0011      D0010 D0011  None    M. Gledhill
   //                        FC18001 — RELEASED FOR USE
   //                          Merge back to master branch
   // 
   //  2022.04.11    001.801   D0010A-000.801   D0010 N/A     D010A   M. Gledhill
   //                        Released for test (SCV)
   // 
   //  2022.04.06    001.101   D0010A-000.104   D0010 N/A     D010A   M. Gledhill
   //                        Comments updated and standardised
   // 
   //  2021.05.22    001.000   D0007      D0006 D0007  None    M. Gledhill
   //                        FC18001 — FORMAL RELEASE FOR USE
   //                          Merge back to master branch
   // 
   //  2021.05.22    001.000   D0006A-001.000   D0006 N/A     D0006A   M. Gledhill
   //                        FC18001 Post-test RELEASED FOR USE
   // 
   //  2021.05.18    000.801   D0006A-000.801   D0006 N/A     D0006A   M. Gledhill
   //                        FC18001 Released for SMT
   // 
   //  2021.05.17    000.101   D0006A-000.101   D0006 N/A     D0006A   M. Gledhill
   //                        FC18001 Migration to VCS
   //  ———————————————————————————————————————————
   //   Where: nnn  =  Major revision
   //         a  =  Type (1-7 Development, 8 Proving, 9 Qualification, 0 Release)
   //       mm  =  Minor revision (must be 00 if a = 0)
   //         Block properties version number should be set to nn.a (only one decimal place)
   // 
   // ▄▄▄▄▄▄▄▄▄▄▄▄▄▄▄▄▄▄▄▄▄▄▄▄▄▄▄▄▄▄▄▄▄▄▄▄▄▄▄▄▄▄▄▄
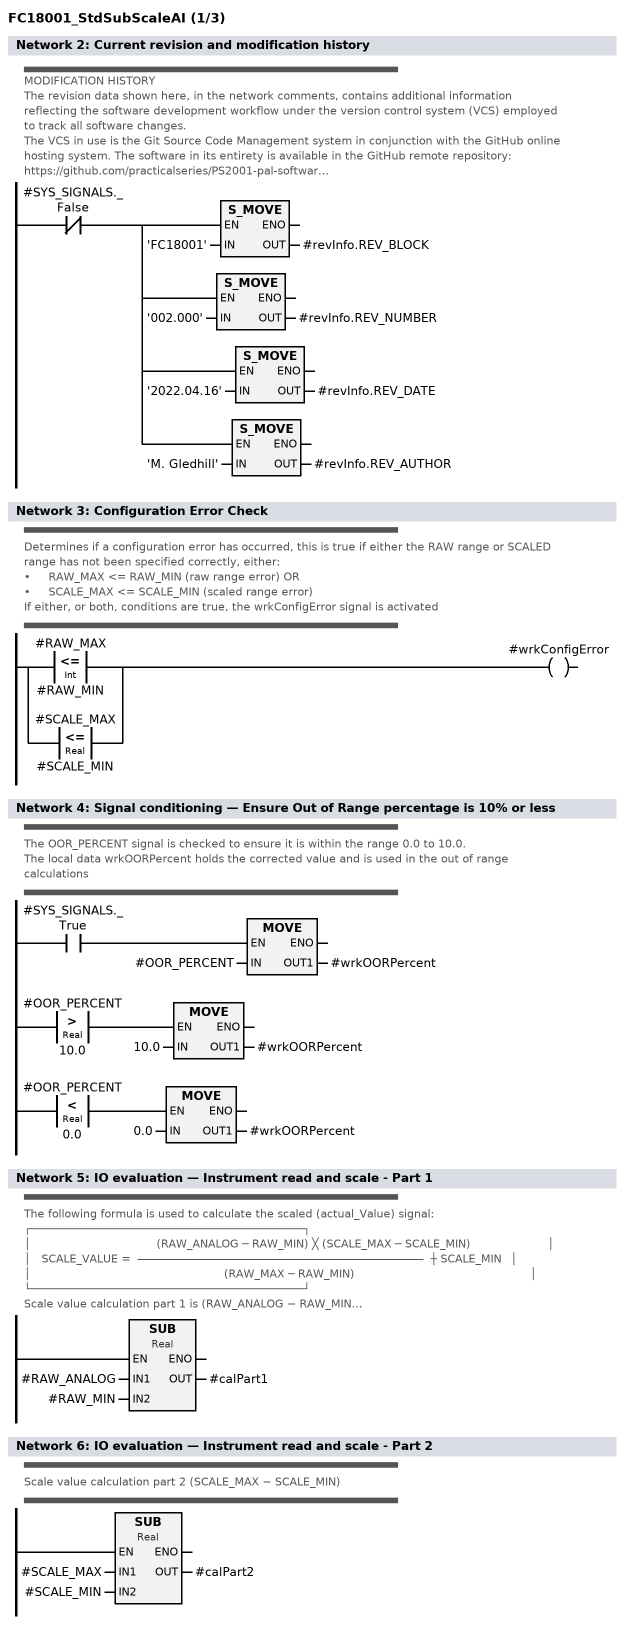
   RUNG wire#powerrail
      I_Contact( #SYS_SIGNALS._False )
      wire#w1
      S_Move(in := 'FC18001', out => #revInfo.REV_BLOCK)
   END_RUNG
   RUNG wire#w1
      S_Move(in := '002.000', out => #revInfo.REV_NUMBER)
   END_RUNG
   RUNG wire#w1
      S_Move(in := '2022.04.16', out => #revInfo.REV_DATE)
   END_RUNG
   RUNG wire#w1
      S_Move(in := 'M. Gledhill', out => #revInfo.REV_AUTHOR)
   END_RUNG
   // the same network as SCL:
   IF NOT #SYS_SIGNALS._False THEN
       #revInfo.REV_BLOCK := 'FC18001';
       #revInfo.REV_NUMBER := '002.000';
       #revInfo.REV_DATE := '2022.04.16';
       #revInfo.REV_AUTHOR := 'M. Gledhill';
   END_IF;
END_REGION

REGION Network 3: Configuration Error Check
   // ▀▀▀▀▀▀▀▀▀▀▀▀▀▀▀▀▀▀▀▀▀▀▀▀▀▀▀▀▀▀▀▀▀▀▀▀▀▀▀▀▀▀▀▀
   // Determines if a configuration error has occurred, this is true if either the RAW range or SCALED 
   // range has not been specified correctly, either:
   // 
   //    •   RAW_MAX <= RAW_MIN (raw range error) OR
   //    •   SCALE_MAX <= SCALE_MIN (scaled range error)
   // 
   // If either, or both, conditions are true, the wrkConfigError signal is activated
   // ▄▄▄▄▄▄▄▄▄▄▄▄▄▄▄▄▄▄▄▄▄▄▄▄▄▄▄▄▄▄▄▄▄▄▄▄▄▄▄▄▄▄▄▄
   RUNG wire#powerrail
      { S7_Templates := "SrcType := Int" } LE_Contact(in1 := #RAW_MAX, in2 := #RAW_MIN)
      wire#w1
      Coil( #wrkConfigError )
   END_RUNG
   RUNG wire#powerrail
      { S7_Templates := "SrcType := Real" } LE_Contact(in1 := #SCALE_MAX, in2 := #SCALE_MIN)
   END_RUNG wire#w1
   // the same network as SCL:
   #wrkConfigError := (#RAW_MAX <= #RAW_MIN) OR (#SCALE_MAX <= #SCALE_MIN);
END_REGION

REGION Network 4: Signal conditioning — Ensure Out of Range percentage is 10% or less
   // ▀▀▀▀▀▀▀▀▀▀▀▀▀▀▀▀▀▀▀▀▀▀▀▀▀▀▀▀▀▀▀▀▀▀▀▀▀▀▀▀▀▀▀▀
   // The OOR_PERCENT signal is checked to ensure it is within the range 0.0 to 10.0.
   // 
   // The local data wrkOORPercent holds the corrected value and is used in the out of range 
   // calculations
   // ▄▄▄▄▄▄▄▄▄▄▄▄▄▄▄▄▄▄▄▄▄▄▄▄▄▄▄▄▄▄▄▄▄▄▄▄▄▄▄▄▄▄▄▄
   RUNG wire#powerrail
      Contact( #SYS_SIGNALS._True )
      Move(in := #OOR_PERCENT, out1 => #wrkOORPercent)
   END_RUNG
   RUNG wire#powerrail
      { S7_Templates := "SrcType := Real" } GT_Contact(in1 := #OOR_PERCENT, in2 := 10.0)
      Move(in := 10.0, out1 => #wrkOORPercent)
   END_RUNG
   RUNG wire#powerrail
      { S7_Templates := "SrcType := Real" } LT_Contact(in1 := #OOR_PERCENT, in2 := 0.0)
      Move(in := 0.0, out1 => #wrkOORPercent)
   END_RUNG
   // the same network as SCL:
   IF #SYS_SIGNALS._True THEN #wrkOORPercent := #OOR_PERCENT; END_IF;
   IF #OOR_PERCENT > 10.0 THEN #wrkOORPercent := 10.0; END_IF;
   IF #OOR_PERCENT < 0.0 THEN #wrkOORPercent := 0.0; END_IF;
END_REGION

REGION Network 5: IO evaluation — Instrument read and scale - Part 1
   // ▀▀▀▀▀▀▀▀▀▀▀▀▀▀▀▀▀▀▀▀▀▀▀▀▀▀▀▀▀▀▀▀▀▀▀▀▀▀▀▀▀▀▀▀
   // The following formula is used to calculate the scaled (actual_Value) signal:
   // ┌──────────────────────────────────────────┐
   // │                                    (RAW_ANALOG ─ RAW_MIN) ╳ (SCALE_MAX ─ SCALE_MIN)          │
   // │ SCALE_VALUE =  ――――――――――――――――――――――――――  ┼ SCALE_MIN   │
   // │                                    (RAW_MAX ─ RAW_MIN)                  │
   // └──────────────────────────────────────────┘
   // 
   // Scale value calculation part 1 is (RAW_ANALOG − RAW_MIN)
   // ▄▄▄▄▄▄▄▄▄▄▄▄▄▄▄▄▄▄▄▄▄▄▄▄▄▄▄▄▄▄▄▄▄▄▄▄▄▄▄▄▄▄▄▄
   RUNG wire#powerrail
      { S7_Templates := "SrcType := Real"; S7_GenerateENO := "TRUE" } Sub(in1 := #RAW_ANALOG, in2 := #RAW_MIN, out => #calPart1)
   END_RUNG
   // the same network as SCL:
   #calPart1 := #RAW_ANALOG - #RAW_MIN;
END_REGION

REGION Network 6: IO evaluation — Instrument read and scale - Part 2
   // ▀▀▀▀▀▀▀▀▀▀▀▀▀▀▀▀▀▀▀▀▀▀▀▀▀▀▀▀▀▀▀▀▀▀▀▀▀▀▀▀▀▀▀▀
   // Scale value calculation part 2 (SCALE_MAX − SCALE_MIN)
   // ▄▄▄▄▄▄▄▄▄▄▄▄▄▄▄▄▄▄▄▄▄▄▄▄▄▄▄▄▄▄▄▄▄▄▄▄▄▄▄▄▄▄▄▄
   RUNG wire#powerrail
      { S7_Templates := "SrcType := Real"; S7_GenerateENO := "TRUE" } Sub(in1 := #SCALE_MAX, in2 := #SCALE_MIN, out => #calPart2)
   END_RUNG
   // the same network as SCL:
   #calPart2 := #SCALE_MAX - #SCALE_MIN;
END_REGION

REGION Network 7: IO evaluation — Instrument read and scale - Part 3
   // ▀▀▀▀▀▀▀▀▀▀▀▀▀▀▀▀▀▀▀▀▀▀▀▀▀▀▀▀▀▀▀▀▀▀▀▀▀▀▀▀▀▀▀▀
   // Scale value calculation part 3 (RAW_MAX − RAW_MIN)
   // 
   // Note:    To prevent inconsistencies and divide by zero errors, if a configuration error is present
   //      (resulting from incorrect range data and indicated by status_ConfigError = TRUE), the
   //      denominator of the calculation (CalPart3) is set to 3.402823 × 1038 (i.e. a very large 
   //      number), the result of this is that the  SCALE_VALUE will equal SCALE_MIN for 
   //      all permitted values of RAW_ANALOG.
   // ▄▄▄▄▄▄▄▄▄▄▄▄▄▄▄▄▄▄▄▄▄▄▄▄▄▄▄▄▄▄▄▄▄▄▄▄▄▄▄▄▄▄▄▄
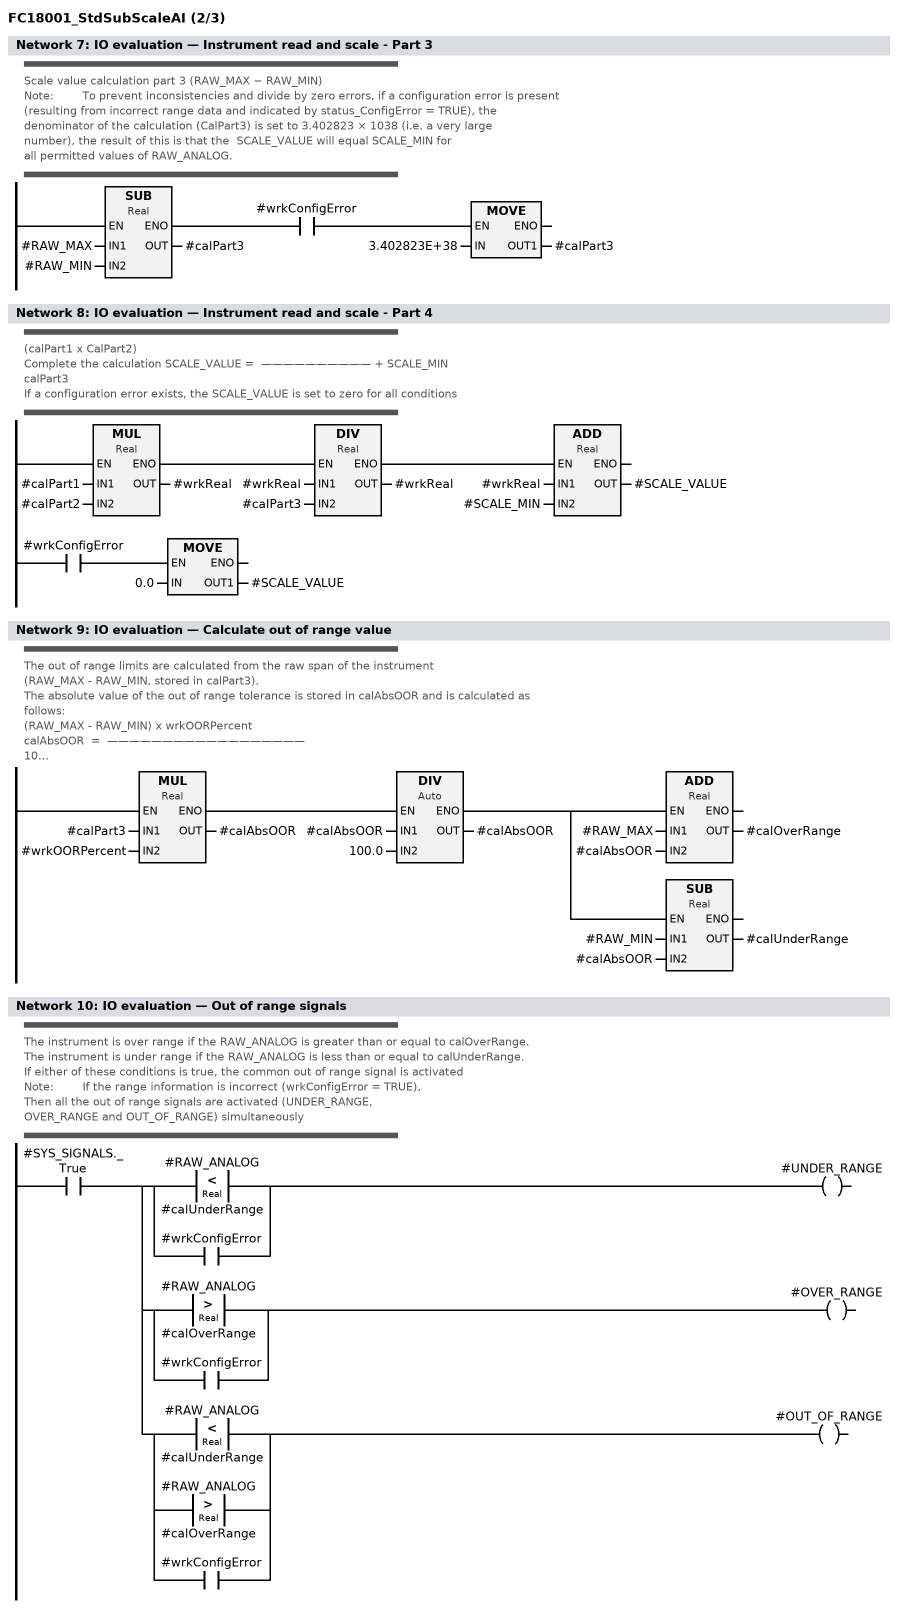
   RUNG wire#powerrail
      { S7_Templates := "SrcType := Real"; S7_GenerateENO := "TRUE" } Sub(in1 := #RAW_MAX, in2 := #RAW_MIN, out => #calPart3)
      Contact( #wrkConfigError )
      Move(in := 3.402823E+38, out1 => #calPart3)
   END_RUNG
   // the same network as SCL:
   // ENO of a box is taken as its EN; it also drops when the box reports an error
   #calPart3 := #RAW_MAX - #RAW_MIN;
   IF #wrkConfigError THEN #calPart3 := 3.402823E+38; END_IF;
END_REGION

REGION Network 8: IO evaluation — Instrument read and scale - Part 4
   // ▀▀▀▀▀▀▀▀▀▀▀▀▀▀▀▀▀▀▀▀▀▀▀▀▀▀▀▀▀▀▀▀▀▀▀▀▀▀▀▀▀▀▀▀
   //                                                                              (calPart1 x CalPart2)
   // Complete the calculation SCALE_VALUE =  —————————— + SCALE_MIN
   //                                                                                         calPart3
   // 
   // If a configuration error exists, the SCALE_VALUE is set to zero for all conditions
   // ▄▄▄▄▄▄▄▄▄▄▄▄▄▄▄▄▄▄▄▄▄▄▄▄▄▄▄▄▄▄▄▄▄▄▄▄▄▄▄▄▄▄▄▄
   RUNG wire#powerrail
      { S7_Templates := "SrcType := Real"; S7_GenerateENO := "TRUE" } Mul(in1 := #calPart1, in2 := #calPart2, out => #wrkReal)
      { S7_Templates := "SrcType := Real"; S7_GenerateENO := "TRUE" } Div(in1 := #wrkReal, in2 := #calPart3, out => #wrkReal)
      { S7_Templates := "SrcType := Real"; S7_GenerateENO := "TRUE" } Add(in1 := #wrkReal, in2 := #SCALE_MIN, out => #SCALE_VALUE)
   END_RUNG
   RUNG wire#powerrail
      Contact( #wrkConfigError )
      Move(in := 0.0, out1 => #SCALE_VALUE)
   END_RUNG
   // the same network as SCL:
   // ENO of a box is taken as its EN; it also drops when the box reports an error
   #wrkReal := #calPart1 * #calPart2;
   #wrkReal := #wrkReal / #calPart3;
   #SCALE_VALUE := #wrkReal + #SCALE_MIN;
   IF #wrkConfigError THEN #SCALE_VALUE := 0.0; END_IF;
END_REGION

REGION Network 9: IO evaluation — Calculate out of range value
   // ▀▀▀▀▀▀▀▀▀▀▀▀▀▀▀▀▀▀▀▀▀▀▀▀▀▀▀▀▀▀▀▀▀▀▀▀▀▀▀▀▀▀▀▀
   // The out of range limits are calculated from the raw span of the instrument 
   // (RAW_MAX - RAW_MIN, stored in calPart3).
   // 
   // The absolute value of the out of range tolerance is stored in calAbsOOR and is calculated as
   // follows:
   // 
   // 
   //                             (RAW_MAX - RAW_MIN) x wrkOORPercent
   // calAbsOOR  =  ——————————————————
   //                                                              100
   // 
   // OR
   // 
   //                             calPart3 x wrkOORPercent
   // calAbsOOR  =  ————————————
   //                                               100
   // 
   // 
   // The instrument is over range if the RAW_ANALOG exceeds RAW_MAX + calAbsOOR 
   // 
   // The instrument is under range if the RAW_ANALOG is less than RAW_MIN - calAbsOOR 
   // ▄▄▄▄▄▄▄▄▄▄▄▄▄▄▄▄▄▄▄▄▄▄▄▄▄▄▄▄▄▄▄▄▄▄▄▄▄▄▄▄▄▄▄▄
   RUNG wire#powerrail
      { S7_Templates := "SrcType := Real"; S7_GenerateENO := "TRUE" } Mul(in1 := #calPart3, in2 := #wrkOORPercent, out => #calAbsOOR)
      Div(in1 := #calAbsOOR, in2 := 100.0, out => #calAbsOOR)
      wire#w1
      { S7_Templates := "SrcType := Real"; S7_GenerateENO := "TRUE" } Add(in1 := #RAW_MAX, in2 := #calAbsOOR, out => #calOverRange)
   END_RUNG
   RUNG wire#w1
      { S7_Templates := "SrcType := Real"; S7_GenerateENO := "TRUE" } Sub(in1 := #RAW_MIN, in2 := #calAbsOOR, out => #calUnderRange)
   END_RUNG
   // the same network as SCL:
   // ENO of a box is taken as its EN; it also drops when the box reports an error
   #calAbsOOR := #calPart3 * #wrkOORPercent;
   #calAbsOOR := #calAbsOOR / 100.0;
   #calOverRange := #RAW_MAX + #calAbsOOR;
   #calUnderRange := #RAW_MIN - #calAbsOOR;
END_REGION

REGION Network 10: IO evaluation — Out of range signals
   // ▀▀▀▀▀▀▀▀▀▀▀▀▀▀▀▀▀▀▀▀▀▀▀▀▀▀▀▀▀▀▀▀▀▀▀▀▀▀▀▀▀▀▀▀
   // The instrument is over range if the RAW_ANALOG is greater than or equal to calOverRange.
   // 
   // The instrument is under range if the RAW_ANALOG is less than or equal to calUnderRange.
   // 
   // If either of these conditions is true, the common out of range signal is activated
   // 
   // Note:    If the range information is incorrect (wrkConfigError = TRUE),
   //      Then all the out of range signals are activated (UNDER_RANGE, 
   //      OVER_RANGE and OUT_OF_RANGE) simultaneously
   // ▄▄▄▄▄▄▄▄▄▄▄▄▄▄▄▄▄▄▄▄▄▄▄▄▄▄▄▄▄▄▄▄▄▄▄▄▄▄▄▄▄▄▄▄
   RUNG wire#powerrail
      Contact( #SYS_SIGNALS._True )
      wire#w1
      { S7_Templates := "SrcType := Real" } LT_Contact(in1 := #RAW_ANALOG, in2 := #calUnderRange)
      wire#w2
      Coil( #UNDER_RANGE )
   END_RUNG
   RUNG wire#w1
      Contact( #wrkConfigError )
   END_RUNG wire#w2
   RUNG wire#w1
      { S7_Templates := "SrcType := Real" } GT_Contact(in1 := #RAW_ANALOG, in2 := #calOverRange)
      wire#w3
      Coil( #OVER_RANGE )
   END_RUNG
   RUNG wire#w1
      Contact( #wrkConfigError )
   END_RUNG wire#w3
   RUNG wire#w1
      { S7_Templates := "SrcType := Real" } LT_Contact(in1 := #RAW_ANALOG, in2 := #calUnderRange)
      wire#w4
      Coil( #OUT_OF_RANGE )
   END_RUNG
   RUNG wire#w1
      { S7_Templates := "SrcType := Real" } GT_Contact(in1 := #RAW_ANALOG, in2 := #calOverRange)
   END_RUNG wire#w4
   RUNG wire#w1
      Contact( #wrkConfigError )
   END_RUNG wire#w4
   // the same network as SCL:
   #UNDER_RANGE := #SYS_SIGNALS._True AND ((#RAW_ANALOG < #calUnderRange) OR #wrkConfigError);
   #OVER_RANGE := #SYS_SIGNALS._True AND ((#RAW_ANALOG > #calOverRange) OR #wrkConfigError);
   #OUT_OF_RANGE := #SYS_SIGNALS._True AND ((#RAW_ANALOG < #calUnderRange) OR (#RAW_ANALOG > #calOverRange) OR #wrkConfigError);
END_REGION

REGION Network 11: LICENCE AND CONTACT INFORMATION
   // ▀▀▀▀▀▀▀▀▀▀▀▀▀▀▀▀▀▀▀▀▀▀▀▀▀▀▀▀▀▀▀▀▀▀▀▀▀▀▀▀▀▀▀▀
   // LICENCE AND CONTACT INFORMATION
   // 
   // This software and its associated documentation is made available under the MIT Licence:
   // 
   // ════════════════════════════════════════════
   // 
   // The MIT License (MIT)
   // 
   // Copyright © 2020 Michael Gledhill
   // 
   // Permission is hereby granted, free of charge, to any person obtaining a copy of this software 
   // and associated documentation files (the “Software”), to deal in the Software without restriction, 
   // including without limitation the rights to use, copy, modify, merge, publish, distribute, 
   // sublicense, and/or sell copies of the Software, and to permit persons to whom the Software is 
   // furnished to do so, subject to the following conditions: 
   // 
   // The above copyright notice and this permission notice shall be included in all copies or 
   // substantial portions of the Software.
   // 
   // THE SOFTWARE IS PROVIDED “AS IS”, WITHOUT WARRANTY OF ANY KIND, EXPRESS OR IMPLIED, 
   // INCLUDING BUT NOT LIMITED TO THE WARRANTIES OF MERCHANTABILITY, FITNESS FOR A 
   // PARTICULAR PURPOSE AND NON-INFRINGEMENT. IN NO EVENT SHALL THE AUTHORS OR COPYRIGHT 
   // HOLDERS BE LIABLE FOR ANY CLAIM, DAMAGES OR OTHER LIABILITY, WHETHER IN AN ACTION OF 
   // CONTRACT, TORT OR OTHERWISE, ARISING FROM, OUT OF OR IN CONNECTION WITH THE SOFTWARE 
   // OR THE USE OR OTHER DEALINGS IN THE SOFTWARE.
   // 
   // ════════════════════════════════════════════
   //                    ┌────────────┐
   // You can reach the author by email here:   │  mg@practicalseries.com  │
   //                    └────────────┘
   // Questions, corrections, constructive criticism and complaints (polite ones) are invited.
   // 
   // ▄▄▄▄▄▄▄▄▄▄▄▄▄▄▄▄▄▄▄▄▄▄▄▄▄▄▄▄▄▄▄▄▄▄▄▄▄▄▄▄▄▄▄▄
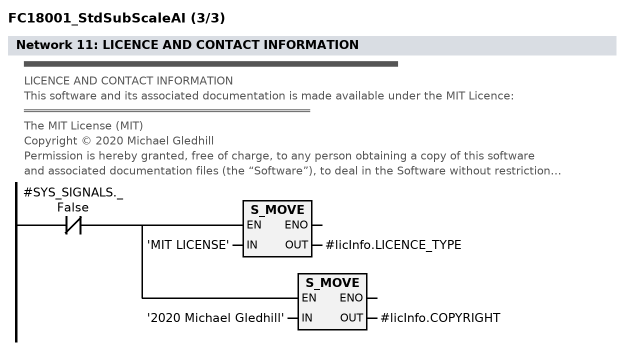
   RUNG wire#powerrail
      I_Contact( #SYS_SIGNALS._False )
      wire#w1
      S_Move(in := 'MIT LICENSE', out => #licInfo.LICENCE_TYPE)
   END_RUNG
   RUNG wire#w1
      S_Move(in := '2020 Michael Gledhill', out => #licInfo.COPYRIGHT)
   END_RUNG
   // the same network as SCL:
   IF NOT #SYS_SIGNALS._False THEN
       #licInfo.LICENCE_TYPE := 'MIT LICENSE';
       #licInfo.COPYRIGHT := '2020 Michael Gledhill';
   END_IF;
END_REGION
END_FUNCTION

FUNCTION "FC18002_StdSubScaleAQ" : Void   // FC18002, LAD
TITLE = Standard Module [SUBROUTINE] — Analog Output Scale
{ S7_Optimized_Access := 'TRUE' }
AUTHOR : M_Gledhill
FAMILY : Subroutine
NAME : StdSubScaleAQ
VERSION : 0.8
// PRACTICAL SERIES AUTOMATION LIBRARY (PAL)   —   COPYRIGHT 2020 – M. GLEDHILL (MIT LICENCE)
//                   ———— ◆ ————
// FULL ONLINE DOCUMENTATION IS AVAILABLE AT: https://practicalseries.com/2001-pal/index.html
// stored: AutoNumber false, IsIECCheckEnabled true, SetENOAutomatically false, UDAEnableTagReadback false
   VAR_INPUT
      AQ_SCALE_SIGNAL : Real;   // Scaled Input
      AQ_RAW_DATA : "UT00802_St_ConstAqRawData";   // Analog Output Signal — raw range and configuration data
      AQ_SCALE_DATA : "UT00852_Sy_ConstAqScaleData";   // Analog Output Signal — scaled range and configuration data
   END_VAR
   VAR_OUTPUT
      AQ_RAW_SIGNAL : Int;   // Actual Output (as an integer for output card)
      OVER_RANGE : Bool;   // Signal Fault - Over range
      UNDER_RANGE : Bool;   // Signal Fault - Under range
      OUT_OF_RANGE : Bool;   // Signal Fault - Out of Range (either over or under)
   END_VAR
   VAR_TEMP
      revInfo : "UT01000_St_SysRevision";   // Revision information for this block
      licInfo : "UT01001_St_SysLicence";   // Licence information for this block
      calPart1 : Real;   // Raw value calculation part 1 (AQ_SCALE_VALUE − SCALE_MIN)
      calPart2 : Real;   // Raw value calculation part 2 (SCALE_MAX − SCALE_MIN)
      calPart3 : Real;   // Raw value calculation part 1 (RAW_MAX − RAW_MIN)
      wrkLimitUnder : Real;   // Actual LIMIT_UNDER in use
      wrkLimitOver : Real;   // Actual LIMIT_OVER in use
      wrkConfigError : Bool;   // Working configuration error exists
      wrkReal : Real;   // Working storage (real)
   END_VAR
BEGIN

